KUKA KRL program: MyProgram_038().src

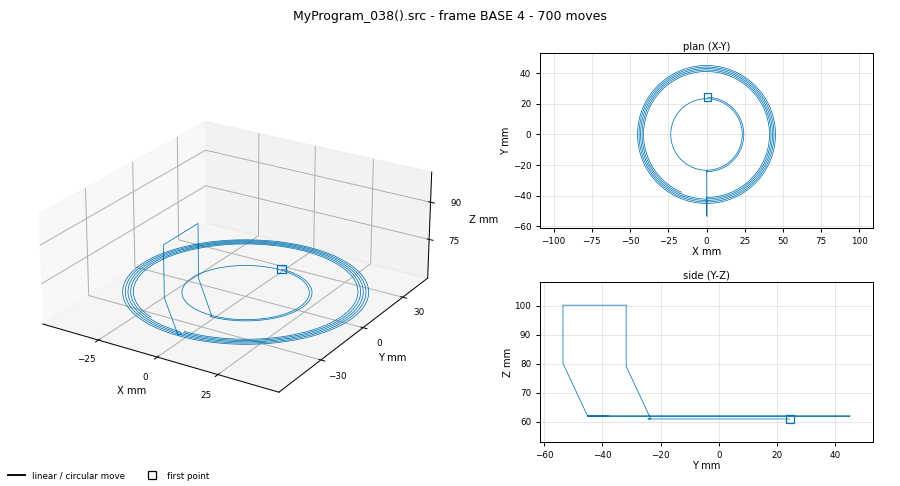
[picture p0: tool path of MyProgram_038().src in frame BASE 4, 700 of 700 moves have a stored position in this frame; points joined in program order, loops and branches not executed]
&ACCESS RVP
&REL 1
&PARAM TEMPLATE = C:\KRC\Roboter\Template\vorgabe
&PARAM EDITMASK = *
DEF MyProgram_038()
; ---- Setting reference (Base) ----
$BASE = BASE_DATA[4]

; --------------------------
; ---- Setting tool (TCP) ----
$TOOL = TOOL_DATA[3]
; --------------------------

$VEL.CP = VEL_APROX_PRINT
Startdeposition()
$VEL.CP = VEL_PRINT
LIN {X 0.6576,Y 24.378,Z 61,A 79.6841,B 24.798,C -3.2768,E1 25.0073,E2 -357.1342} C_DIS
LIN {X 2.4777,Y 24.2605,Z 61,A 75.3476,B 24.798,C -3.2762,E1 25.0194,E2 -352.7985} C_DIS
LIN {X 4.2079,Y 24.0211,Z 61,A 71.1898,B 24.7983,C -3.2745,E1 25.0308,E2 -348.6408} C_DIS
LIN {X 6.0369,Y 23.6276,Z 61,A 66.8091,B 24.7986,C -3.2723,E1 25.0427,E2 -344.261} C_DIS
LIN {X 7.8263,Y 23.0968,Z 61,A 62.2092,B 24.7992,C -3.2672,E1 25.055,E2 -339.6573} C_DIS
LIN {X 9.7348,Y 22.3594,Z 61,A 57.8843,B 24.7992,C -3.2666,E1 25.0661,E2 -335.3411} C_DIS
LIN {X 11.6331,Y 21.4331,Z 61,A 51.9674,B 24.8011,C -3.2518,E1 25.0809,E2 -329.4051} C_DIS
LIN {X 13.7357,Y 20.1506,Z 61,A 46.5226,B 24.8018,C -3.2461,E1 25.0936,E2 -323.9647} C_DIS
LIN {X 15.5109,Y 18.8183,Z 61,A 41.6965,B 24.8025,C -3.2406,E1 25.1042,E2 -319.1435} C_DIS
LIN {X 16.7453,Y 17.7285,Z 61,A 37.3106,B 24.804,C -3.2279,E1 25.1132,E2 -314.7453} C_DIS
LIN {X 18.8106,Y 15.5203,Z 61,A 30.4494,B 24.8056,C -3.2147,E1 25.1259,E2 -307.8835} C_DIS
LIN {X 20.1422,Y 13.748,Z 61,A 25.5563,B 24.8068,C -3.2054,E1 25.1338,E2 -302.992} C_DIS
LIN {X 20.9302,Y 12.5161,Z 61,A 22.3998,B 24.8075,C -3.1995,E1 25.1384,E2 -299.8377} C_DIS
LIN {X 21.6103,Y 11.3009,Z 61,A 18.8323,B 24.8089,C -3.1877,E1 25.1432,E2 -296.2609} C_DIS
LIN {X 22.463,Y 9.4933,Z 61,A 14.3404,B 24.8102,C -3.1769,E1 25.1483,E2 -291.768} C_DIS
LIN {X 23.0782,Y 7.8813,Z 61,A 10.2587,B 24.8116,C -3.165,E1 25.1522,E2 -287.6809} C_DIS
LIN {X 23.5913,Y 6.1782,Z 61,A 6.2664,B 24.8129,C -3.1548,E1 25.1552,E2 -283.6871} C_DIS
LIN {X 23.9107,Y 4.794,Z 61,A 3.2615,B 24.8136,C -3.1484,E1 25.157,E2 -280.6846} C_DIS
LIN {X 24.0965,Y 3.7504,Z 61,A 0.195,B 24.8153,C -3.1345,E1 25.1584,E2 -277.6031} C_DIS
LIN {X 24.3261,Y 1.7192,Z 61,A -4.4464,B 24.8168,C -3.1214,E1 25.1596,E2 -272.9583} C_DIS
LIN {X 24.3856,Y -0.076,Z 61,A -8.4621,B 24.8181,C -3.1105,E1 25.1597,E2 -268.9408} C_DIS
LIN {X 24.3156,Y -1.8616,Z 61,A -12.7948,B 24.8198,C -3.0959,E1 25.1591,E2 -264.5991} C_DIS
LIN {X 24.1022,Y -3.7139,Z 61,A -16.7586,B 24.8209,C -3.0869,E1 25.1576,E2 -260.6373} C_DIS
LIN {X 23.6477,Y -5.9589,Z 61,A -22.4108,B 24.8231,C -3.0672,E1 25.1543,E2 -254.9714} C_DIS
LIN {X 23.2604,Y -7.3264,Z 61,A -26.4458,B 24.8252,C -3.0494,E1 25.1509,E2 -250.9172} C_DIS
LIN {X 22.4045,Y -9.6314,Z 61,A -31.5534,B 24.8263,C -3.0395,E1 25.1457,E2 -245.8144} C_DIS
LIN {X 21.5556,Y -11.4048,Z 61,A -36.5253,B 24.8283,C -3.0224,E1 25.1394,E2 -240.8283} C_DIS
LIN {X 20.2637,Y -13.5686,Z 61,A -41.8677,B 24.8295,C -3.0122,E1 25.1315,E2 -235.4888} C_DIS
LIN {X 19.4766,Y -14.6755,Z 61,A -44.8622,B 24.8302,C -3.0059,E1 25.1265,E2 -232.4937} C_DIS
LIN {X 18.4591,Y -15.9371,Z 61,A -49.0447,B 24.8317,C -2.9922,E1 25.119,E2 -228.2982} C_DIS
LIN {X 17.1878,Y -17.3001,Z 61,A -53.3461,B 24.8328,C -2.9826,E1 25.1107,E2 -223.9923} C_DIS
LIN {X 15.9747,Y -18.4257,Z 61,A -56.7982,B 24.8333,C -2.9783,E1 25.1035,E2 -220.5439} C_DIS
LIN {X 15.0855,Y -19.1609,Z 61,A -59.5057,B 24.8339,C -2.9725,E1 25.0976,E2 -217.8329} C_DIS
LIN {X 13.9507,Y -20.0022,Z 61,A -63.1749,B 24.8351,C -2.9623,E1 25.0893,E2 -214.1524} C_DIS
LIN {X 12.5585,Y -20.9047,Z 61,A -66.515,B 24.8353,C -2.9606,E1 25.0814,E2 -210.819} C_DIS
LIN {X 11.549,Y -21.4787,Z 61,A -69.6521,B 24.8362,C -2.952,E1 25.0737,E2 -207.6705} C_DIS
LIN {X 10.141,Y -22.1785,Z 61,A -73.5285,B 24.8371,C -2.9445,E1 25.0639,E2 -203.7865} C_DIS
LIN {X 8.4683,Y -22.8694,Z 61,A -77.5795,B 24.8375,C -2.9407,E1 25.0534,E2 -199.7352} C_DIS
LIN {X 7.2197,Y -23.2934,Z 61,A -80.9229,B 24.8381,C -2.9348,E1 25.0445,E2 -196.3842} C_DIS
LIN {X 5.8698,Y -23.6699,Z 61,A -84.8468,B 24.8391,C -2.926,E1 25.0338,E2 -192.4451} C_DIS
LIN {X 3.4157,Y -24.1463,Z 61,A -89.8947,B 24.8388,C -2.9287,E1 25.0199,E2 -187.4091} C_DIS
LIN {X 1.6154,Y -24.3331,Z 61,A -94.2888,B 24.8392,C -2.9255,E1 25.0077,E2 -183.0095} C_DIS
LIN {X 0.1346,Y -24.3815,Z 61,A -96.6732,B 24.8383,C -2.9336,E1 25.0011,E2 -180.645} C_DIS
Enddeposition()
LIN {X 0.1346,Y -24.3815,Z 61,A -96.6732,B 24.8383,C -2.9336,E1 25.0011,E2 -180.645} C_DIS
Startdeposition()
$VEL.CP = VEL_PRINT
LIN {X 0.4821,Y -23.3967,Z 61,A -94.7836,B 24.8354,C -2.9592,E1 25.0065,E2 -182.5952} C_DIS
LIN {X 2.1977,Y -23.2983,Z 61,A -90.4932,B 24.8351,C -2.9619,E1 25.0185,E2 -186.8898} C_DIS
LIN {X 3.9008,Y -23.0743,Z 61,A -86.3802,B 24.8349,C -2.964,E1 25.0299,E2 -191.004} C_DIS
LIN {X 5.5815,Y -22.7263,Z 61,A -82.17,B 24.8345,C -2.9679,E1 25.0413,E2 -195.2177} C_DIS
LIN {X 7.3446,Y -22.2197,Z 61,A -77.7872,B 24.834,C -2.972,E1 25.053,E2 -199.6024} C_DIS
LIN {X 8.8729,Y -21.6544,Z 61,A -73.7272,B 24.8333,C -2.978,E1 25.0636,E2 -203.6678} C_DIS
LIN {X 10.4384,Y -20.9447,Z 61,A -69.5097,B 24.8326,C -2.9846,E1 25.0742,E2 -207.8899} C_DIS
LIN {X 11.9544,Y -20.1179,Z 61,A -65.2481,B 24.8317,C -2.9923,E1 25.0846,E2 -212.1571} C_DIS
LIN {X 13.4495,Y -19.151,Z 61,A -60.9988,B 24.8309,C -2.9996,E1 25.0944,E2 -216.4095} C_DIS
LIN {X 14.8782,Y -18.0634,Z 61,A -56.5009,B 24.8297,C -3.0099,E1 25.1043,E2 -220.9151} C_DIS
LIN {X 16.2712,Y -16.8192,Z 61,A -51.9607,B 24.8286,C -3.0201,E1 25.1136,E2 -225.4608} C_DIS
LIN {X 17.5911,Y -15.4335,Z 61,A -47.3398,B 24.8273,C -3.0309,E1 25.1223,E2 -230.087} C_DIS
LIN {X 18.7335,Y -14.0247,Z 61,A -42.9703,B 24.8261,C -3.0417,E1 25.1298,E2 -234.4614} C_DIS
LIN {X 19.7022,Y -12.6277,Z 61,A -38.7961,B 24.8248,C -3.0531,E1 25.1363,E2 -238.642} C_DIS
LIN {X 20.5911,Y -11.1195,Z 61,A -34.493,B 24.8234,C -3.0654,E1 25.1422,E2 -242.9519} C_DIS
LIN {X 21.2756,Y -9.747,Z 61,A -30.8472,B 24.8222,C -3.0752,E1 25.1465,E2 -246.6012} C_DIS
LIN {X 21.9018,Y -8.2431,Z 61,A -26.7916,B 24.8208,C -3.0878,E1 25.1507,E2 -250.6643} C_DIS
LIN {X 22.4767,Y -6.5158,Z 61,A -22.4671,B 24.8193,C -3.0999,E1 25.1543,E2 -254.9928} C_DIS
LIN {X 22.8784,Y -4.9215,Z 61,A -18.4694,B 24.8179,C -3.112,E1 25.1568,E2 -258.9961} C_DIS
LIN {X 23.1776,Y -3.2307,Z 61,A -14.2077,B 24.8163,C -3.1258,E1 25.1587,E2 -263.2653} C_DIS
LIN {X 23.3521,Y -1.5221,Z 61,A -10.0343,B 24.8148,C -3.1386,E1 25.1596,E2 -267.4442} C_DIS
LIN {X 23.3967,Y 0.4812,Z 61,A -5.2469,B 24.8131,C -3.1525,E1 25.1596,E2 -272.2363} C_DIS
LIN {X 23.2984,Y 2.1957,Z 61,A -0.9845,B 24.8115,C -3.1662,E1 25.1587,E2 -276.5057} C_DIS
LIN {X 23.0748,Y 3.8974,Z 61,A 3.1273,B 24.8101,C -3.178,E1 25.157,E2 -280.6214} C_DIS
LIN {X 22.7212,Y 5.6026,Z 61,A 7.3368,B 24.8086,C -3.1902,E1 25.1544,E2 -284.8353} C_DIS
LIN {X 22.2215,Y 7.3391,Z 61,A 11.6522,B 24.8072,C -3.2019,E1 25.1509,E2 -289.1539} C_DIS
LIN {X 21.684,Y 8.8002,Z 61,A 15.6019,B 24.8057,C -3.2142,E1 25.1469,E2 -293.1108} C_DIS
LIN {X 20.9488,Y 10.43,Z 61,A 19.8688,B 24.8044,C -3.225,E1 25.1417,E2 -297.3802} C_DIS
LIN {X 20.117,Y 11.9559,Z 61,A 24.1861,B 24.803,C -3.2367,E1 25.1358,E2 -301.703} C_DIS
LIN {X 19.0819,Y 13.547,Z 61,A 28.7529,B 24.8017,C -3.2473,E1 25.1286,E2 -306.2725} C_DIS
LIN {X 17.9987,Y 14.9561,Z 61,A 33.0946,B 24.8004,C -3.2573,E1 25.121,E2 -310.6175} C_DIS
LIN {X 16.7652,Y 16.3272,Z 61,A 37.6578,B 24.7992,C -3.2674,E1 25.1123,E2 -315.1848} C_DIS
LIN {X 15.4284,Y 17.5955,Z 61,A 42.0949,B 24.7982,C -3.2755,E1 25.1031,E2 -319.6232} C_DIS
LIN {X 14.0165,Y 18.7397,Z 61,A 46.481,B 24.7973,C -3.2827,E1 25.0935,E2 -324.0102} C_DIS
LIN {X 12.599,Y 19.7207,Z 61,A 50.7583,B 24.7964,C -3.2898,E1 25.0835,E2 -328.2902} C_DIS
LIN {X 11.0488,Y 20.6295,Z 61,A 55.0577,B 24.7958,C -3.2948,E1 25.0731,E2 -332.5889} C_DIS
LIN {X 9.4872,Y 21.3927,Z 61,A 59.3098,B 24.7952,C -3.2996,E1 25.0623,E2 -336.8416} C_DIS
LIN {X 7.8909,Y 22.0315,Z 61,A 63.4425,B 24.7948,C -3.3028,E1 25.0515,E2 -340.973} C_DIS
LIN {X 6.2392,Y 22.555,Z 61,A 67.7455,B 24.7943,C -3.3063,E1 25.04,E2 -345.2768} C_DIS
LIN {X 4.5669,Y 22.9521,Z 61,A 71.9513,B 24.7941,C -3.3083,E1 25.0285,E2 -349.4818} C_DIS
LIN {X 2.9587,Y 23.2139,Z 61,A 76.0249,B 24.7939,C -3.31,E1 25.0173,E2 -353.5558} C_DIS
LIN {X 1.1581,Y 23.3733,Z 61,A 80.3651,B 24.7939,C -3.3094,E1 25.0052,E2 -357.8926} C_DIS
LIN {X -0.4696,Y 23.397,Z 61,A 84.3727,B 24.794,C -3.3087,E1 24.994,E2 -361.8986} C_DIS
LIN {X -2.2037,Y 23.2977,Z 61,A 88.6974,B 24.7942,C -3.3074,E1 24.982,E2 -366.2221} C_DIS
LIN {X -3.9081,Y 23.073,Z 61,A 92.8279,B 24.7946,C -3.3041,E1 24.9706,E2 -370.3482} C_DIS
LIN {X -5.5911,Y 22.724,Z 61,A 97.0452,B 24.7951,C -3.3005,E1 24.9591,E2 -374.5623} C_DIS
LIN {X -7.3245,Y 22.2262,Z 61,A 101.4177,B 24.7957,C -3.2953,E1 24.9474,E2 -378.93} C_DIS
LIN {X -8.8731,Y 21.6543,Z 61,A 105.5215,B 24.7963,C -3.2905,E1 24.9368,E2 -383.0309} C_DIS
LIN {X -10.4256,Y 20.951,Z 61,A 109.7063,B 24.7971,C -3.2842,E1 24.9262,E2 -387.2115} C_DIS
LIN {X -11.9152,Y 20.1411,Z 61,A 113.9587,B 24.7979,C -3.2778,E1 24.9159,E2 -391.4609} C_DIS
LIN {X -13.4405,Y 19.1572,Z 61,A 118.3881,B 24.799,C -3.2692,E1 24.9057,E2 -395.8847} C_DIS
LIN {X -14.9859,Y 17.9739,Z 61,A 123.2373,B 24.8001,C -3.2597,E1 24.8951,E2 -400.7292} C_DIS
LIN {X -16.4031,Y 16.6906,Z 61,A 127.8701,B 24.8015,C -3.2488,E1 24.8857,E2 -405.3548} C_DIS
LIN {X -17.6037,Y 15.419,Z 61,A 132.2093,B 24.8027,C -3.2387,E1 24.8776,E2 -409.6891} C_DIS
LIN {X -18.7457,Y 14.0085,Z 61,A 136.6265,B 24.8041,C -3.2271,E1 24.87,E2 -414.0995} C_DIS
LIN {X -19.7705,Y 12.5213,Z 61,A 141.1344,B 24.8055,C -3.2156,E1 24.8631,E2 -418.6023} C_DIS
LIN {X -20.6499,Y 11.0105,Z 61,A 145.3779,B 24.807,C -3.2033,E1 24.8573,E2 -422.8388} C_DIS
LIN {X -21.3982,Y 9.4747,Z 61,A 149.5929,B 24.8085,C -3.1913,E1 24.8524,E2 -427.048} C_DIS
LIN {X -22.0333,Y 7.886,Z 61,A 153.7349,B 24.81,C -3.1786,E1 24.8483,E2 -431.1828} C_DIS
LIN {X -22.5504,Y 6.2556,Z 61,A 158.034,B 24.8115,C -3.1664,E1 24.8449,E2 -435.4775} C_DIS
LIN {X -22.9461,Y 4.5961,Z 61,A 162.3444,B 24.8129,C -3.1541,E1 24.8423,E2 -439.7839} C_DIS
LIN {X -23.2409,Y 2.7382,Z 61,A 166.9452,B 24.8146,C -3.1398,E1 24.8405,E2 -444.3777} C_DIS
LIN {X -23.3851,Y 0.8879,Z 61,A 171.5741,B 24.8163,C -3.126,E1 24.8398,E2 -449.0015} C_DIS
LIN {X -23.3863,Y -0.8572,Z 61,A 175.7875,B 24.8179,C -3.1124,E1 24.84,E2 -453.2077} C_DIS
LIN {X -23.2682,Y -2.4958,Z 61,A 179.9115,B 24.8193,C -3.1005,E1 24.8411,E2 -457.3279} C_DIS
LIN {X -23.0063,Y -4.2856,Z 61,A -175.7162,B 24.8209,C -3.0868,E1 24.8431,E2 -461.6933} C_DIS
LIN {X -22.6518,Y -5.8766,Z 61,A -171.6959,B 24.8222,C -3.0751,E1 24.8457,E2 -465.709} C_DIS
LIN {X -22.1592,Y -7.5238,Z 61,A -167.406,B 24.8236,C -3.0632,E1 24.8494,E2 -469.9952} C_DIS
LIN {X -21.5076,Y -9.2238,Z 61,A -162.8218,B 24.825,C -3.0514,E1 24.8542,E2 -474.5765} C_DIS
LIN {X -20.9375,Y -10.4529,Z 61,A -159.6322,B 24.8261,C -3.0418,E1 24.8581,E2 -477.7603} C_DIS
LIN {X -20.1157,Y -11.9582,Z 61,A -155.3205,B 24.8273,C -3.0314,E1 24.8641,E2 -482.0699} C_DIS
LIN {X -19.0827,Y -13.5458,Z 61,A -150.6719,B 24.8286,C -3.0201,E1 24.8713,E2 -486.7145} C_DIS
LIN {X -18.0046,Y -14.9489,Z 61,A -146.3168,B 24.8297,C -3.0103,E1 24.8789,E2 -491.0664} C_DIS
LIN {X -16.7508,Y -16.3422,Z 61,A -141.7569,B 24.8308,C -3.0004,E1 24.8876,E2 -495.6225} C_DIS
LIN {X -15.4267,Y -17.597,Z 61,A -137.2275,B 24.8317,C -2.9921,E1 24.897,E2 -500.1504} C_DIS
LIN {X -14.0182,Y -18.7384,Z 61,A -132.8261,B 24.8326,C -2.9841,E1 24.9067,E2 -504.5489} C_DIS
LIN {X -12.5345,Y -19.762,Z 61,A -128.3797,B 24.8334,C -2.9776,E1 24.917,E2 -508.9943} C_DIS
LIN {X -11.0359,Y -20.6365,Z 61,A -124.1142,B 24.834,C -2.9721,E1 24.9274,E2 -513.259} C_DIS
LIN {X -9.4793,Y -21.3962,Z 61,A -119.8794,B 24.8345,C -2.9673,E1 24.9381,E2 -517.493} C_DIS
LIN {X -7.8834,Y -22.0343,Z 61,A -115.7407,B 24.835,C -2.9631,E1 24.9489,E2 -521.6302} C_DIS
LIN {X -6.2449,Y -22.5534,Z 61,A -111.4444,B 24.8352,C -2.9609,E1 24.9604,E2 -525.9284} C_DIS
LIN {X -4.5731,Y -22.9509,Z 61,A -107.2323,B 24.8355,C -2.959,E1 24.9719,E2 -530.1414} C_DIS
LIN {X -2.9659,Y -23.213,Z 61,A -103.1543,B 24.8355,C -2.9589,E1 24.9832,E2 -534.2224} C_DIS
LIN {X -1.147,Y -23.3739,Z 61,A -98.7713,B 24.8355,C -2.9582,E1 24.9954,E2 -538.6054} C_DIS
LIN {X 0.1301,Y -23.3984,Z 61,A -96.7291,B 24.8364,C -2.9502,E1 25.0011,E2 -540.6285} C_DIS
Enddeposition()
LIN {X 0.1399,Y -25.5114,Z 65.5315,A -96.7152,B 24.8371,C -2.9443,E1 25.0011,E2 -540.6285} C_DIS
LIN {X 0.1693,Y -31.8506,Z 79.1262,A -96.6781,B 24.8388,C -2.9287,E1 25.0011,E2 -540.6285} C_DIS
LIN {X 0.1693,Y -31.8506,Z 100.1262,A -97.0269,B 24.8222,C -3.0752,E1 25.0011,E2 -540.6285} C_DIS
LIN {X 0.2145,Y -53.5807,Z 100.1262,A -96.4159,B 24.8624,C -2.7068,E1 25.0003,E2 -540.3627} C_DIS
LIN {X 0.2145,Y -53.5807,Z 80.1262,A -96.0843,B 24.8763,C -2.5674,E1 25.0003,E2 -540.3627} C_DIS
LIN {X 0.2145,Y -47.2414,Z 66.5315,A -96.118,B 24.8749,C -2.5815,E1 25.0003,E2 -540.3627} C_DIS
LIN {X 0.2145,Y -45.1283,Z 62,A -96.1307,B 24.8744,C -2.5869,E1 25.0003,E2 -540.3627} C_DIS
Startdeposition()
$VEL.CP = VEL_PRINT
LIN {X 1.6717,Y -45.1007,Z 62,A -93.3413,B 24.8729,C -2.6023,E1 25.0082,E2 -543.1881} C_DIS
LIN {X 3.8826,Y -44.9643,Z 62,A -90.5016,B 24.8727,C -2.604,E1 25.0161,E2 -546.0305} C_DIS
LIN {X 6.0842,Y -44.7196,Z 62,A -87.7329,B 24.8726,C -2.605,E1 25.0238,E2 -548.7995} C_DIS
LIN {X 8.2712,Y -44.3672,Z 62,A -84.9157,B 24.8724,C -2.6073,E1 25.0315,E2 -551.619} C_DIS
LIN {X 10.428,Y -43.9104,Z 62,A -82.1224,B 24.8721,C -2.6097,E1 25.0392,E2 -554.4144} C_DIS
LIN {X 12.5801,Y -43.3429,Z 62,A -79.3131,B 24.8719,C -2.6124,E1 25.0467,E2 -557.2255} C_DIS
LIN {X 14.6818,Y -42.6769,Z 62,A -76.512,B 24.8715,C -2.6158,E1 25.0542,E2 -560.0294} C_DIS
LIN {X 16.7582,Y -41.905,Z 62,A -73.7082,B 24.8712,C -2.6195,E1 25.0615,E2 -562.8357} C_DIS
LIN {X 18.8037,Y -41.0278,Z 62,A -70.892,B 24.8708,C -2.6235,E1 25.0687,E2 -565.6545} C_DIS
LIN {X 20.7849,Y -40.0607,Z 62,A -68.0934,B 24.8703,C -2.628,E1 25.0756,E2 -568.4562} C_DIS
LIN {X 22.7346,Y -38.9872,Z 62,A -65.2886,B 24.8699,C -2.6326,E1 25.0825,E2 -571.2636} C_DIS
LIN {X 24.6202,Y -37.8247,Z 62,A -62.488,B 24.8694,C -2.6377,E1 25.0891,E2 -574.0671} C_DIS
LIN {X 26.438,Y -36.5773,Z 62,A -59.6921,B 24.8688,C -2.6432,E1 25.0955,E2 -576.8664} C_DIS
LIN {X 28.201,Y -35.236,Z 62,A -56.8931,B 24.8682,C -2.6489,E1 25.1016,E2 -579.6686} C_DIS
LIN {X 29.8959,Y -33.8098,Z 62,A -54.1044,B 24.8677,C -2.6547,E1 25.1075,E2 -582.4602} C_DIS
LIN {X 31.5264,Y -32.2948,Z 62,A -51.2936,B 24.867,C -2.661,E1 25.1132,E2 -585.2743} C_DIS
LIN {X 33.073,Y -30.7089,Z 62,A -48.5064,B 24.8664,C -2.6674,E1 25.1186,E2 -588.0646} C_DIS
LIN {X 34.5333,Y -29.0572,Z 62,A -45.7138,B 24.8657,C -2.6744,E1 25.1237,E2 -590.8609} C_DIS
LIN {X 35.9175,Y -27.3277,Z 62,A -42.918,B 24.865,C -2.6814,E1 25.1285,E2 -593.6602} C_DIS
LIN {X 37.221,Y -25.5237,Z 62,A -40.1096,B 24.8642,C -2.6887,E1 25.133,E2 -596.4722} C_DIS
LIN {X 38.4231,Y -23.6756,Z 62,A -37.328,B 24.8635,C -2.6962,E1 25.1372,E2 -599.2574} C_DIS
LIN {X 39.5435,Y -21.7525,Z 62,A -34.5206,B 24.8627,C -2.7038,E1 25.141,E2 -602.0684} C_DIS
LIN {X 40.5632,Y -19.786,Z 62,A -31.7266,B 24.8619,C -2.7117,E1 25.1445,E2 -604.8661} C_DIS
LIN {X 41.4852,Y -17.7718,Z 62,A -28.9427,B 24.8611,C -2.7195,E1 25.1477,E2 -607.6532} C_DIS
LIN {X 42.3037,Y -15.7247,Z 62,A -26.1532,B 24.8603,C -2.7277,E1 25.1505,E2 -610.4468} C_DIS
LIN {X 43.0274,Y -13.62,Z 62,A -23.3563,B 24.8594,C -2.7358,E1 25.1529,E2 -613.2469} C_DIS
LIN {X 43.6413,Y -11.5025,Z 62,A -20.5675,B 24.8586,C -2.7442,E1 25.155,E2 -616.0397} C_DIS
LIN {X 44.1552,Y -9.337,Z 62,A -17.7713,B 24.8577,C -2.7525,E1 25.1567,E2 -618.8391} C_DIS
LIN {X 44.5586,Y -7.1695,Z 62,A -14.973,B 24.8568,C -2.7612,E1 25.1581,E2 -621.6417} C_DIS
LIN {X 44.8578,Y -4.9641,Z 62,A -12.1768,B 24.8559,C -2.7696,E1 25.159,E2 -624.4411} C_DIS
LIN {X 45.0473,Y -2.757,Z 62,A -9.3942,B 24.8551,C -2.7778,E1 25.1596,E2 -627.2268} C_DIS
LIN {X 45.1183,Y -1.0971,Z 62,A -7.1841,B 24.8542,C -2.7864,E1 25.1598,E2 -629.4439} C_DIS
LIN {X 45.1178,Y 1.1181,Z 62,A -4.498,B 24.8535,C -2.7928,E1 25.1597,E2 -632.1293} C_DIS
LIN {X 45.0094,Y 3.3201,Z 62,A -1.7185,B 24.8526,C -2.8012,E1 25.1592,E2 -634.9121} C_DIS
LIN {X 44.7923,Y 5.5246,Z 62,A 1.0837,B 24.8517,C -2.8097,E1 25.1583,E2 -637.7179} C_DIS
LIN {X 44.4654,Y 7.7261,Z 62,A 3.9908,B 24.8506,C -2.8199,E1 25.157,E2 -640.632} C_DIS
LIN {X 44.0327,Y 9.8986,Z 62,A 6.6733,B 24.85,C -2.826,E1 25.1555,E2 -643.3132} C_DIS
LIN {X 43.494,Y 12.0473,Z 62,A 9.457,B 24.8491,C -2.8338,E1 25.1535,E2 -646.0995} C_DIS
LIN {X 42.8075,Y 14.2943,Z 62,A 12.3147,B 24.8484,C -2.8403,E1 25.151,E2 -648.9562} C_DIS
LIN {X 42.1037,Y 16.2524,Z 62,A 15.0449,B 24.8475,C -2.8494,E1 25.1484,E2 -651.693} C_DIS
LIN {X 41.2555,Y 18.2988,Z 62,A 17.8491,B 24.8466,C -2.8572,E1 25.1453,E2 -654.5} C_DIS
LIN {X 40.3127,Y 20.2917,Z 62,A 20.6475,B 24.8458,C -2.8648,E1 25.1419,E2 -657.3015} C_DIS
LIN {X 39.2633,Y 22.2544,Z 62,A 23.43,B 24.8451,C -2.8715,E1 25.1381,E2 -660.0853} C_DIS
LIN {X 38.1297,Y 24.1453,Z 62,A 26.2223,B 24.8443,C -2.8786,E1 25.134,E2 -662.8801} C_DIS
LIN {X 36.8929,Y 25.9957,Z 62,A 29.0322,B 24.8436,C -2.8853,E1 25.1296,E2 -665.6922} C_DIS
LIN {X 35.5729,Y 27.7747,Z 62,A 31.8295,B 24.8429,C -2.8917,E1 25.1248,E2 -668.4912} C_DIS
LIN {X 34.1741,Y 29.4788,Z 62,A 34.6141,B 24.8422,C -2.8978,E1 25.1198,E2 -671.2776} C_DIS
LIN {X 32.6792,Y 31.1277,Z 62,A 37.4165,B 24.8416,C -2.9034,E1 25.1145,E2 -674.0812} C_DIS
LIN {X 31.1125,Y 32.6937,Z 62,A 40.2159,B 24.841,C -2.909,E1 25.1089,E2 -676.882} C_DIS
LIN {X 29.4788,Y 34.1741,Z 62,A 43.0122,B 24.8404,C -2.9143,E1 25.103,E2 -679.6799} C_DIS
LIN {X 27.7581,Y 35.5858,Z 62,A 45.8169,B 24.8399,C -2.9191,E1 25.0969,E2 -682.4853} C_DIS
LIN {X 25.9872,Y 36.899,Z 62,A 48.6244,B 24.8394,C -2.9239,E1 25.0906,E2 -685.2944} C_DIS
LIN {X 24.1364,Y 38.1352,Z 62,A 51.4212,B 24.8389,C -2.9278,E1 25.084,E2 -688.0912} C_DIS
LIN {X 22.2453,Y 39.2685,Z 62,A 54.2303,B 24.8385,C -2.9319,E1 25.0772,E2 -690.9015} C_DIS
LIN {X 20.2917,Y 40.3127,Z 62,A 57.0342,B 24.8381,C -2.9353,E1 25.0703,E2 -693.7058} C_DIS
LIN {X 18.2796,Y 41.264,Z 62,A 59.8435,B 24.8378,C -2.9382,E1 25.0631,E2 -696.5149} C_DIS
LIN {X 16.2329,Y 42.1113,Z 62,A 62.7796,B 24.8372,C -2.943,E1 25.0555,E2 -699.4558} C_DIS
LIN {X 14.147,Y 42.857,Z 62,A 65.4473,B 24.8372,C -2.943,E1 25.0485,E2 -702.1182} C_DIS
LIN {X 11.9926,Y 43.5089,Z 62,A 68.2784,B 24.8371,C -2.9445,E1 25.0409,E2 -704.9481} C_DIS
LIN {X 9.8884,Y 44.0351,Z 62,A 71.0705,B 24.8368,C -2.9466,E1 25.0333,E2 -707.7412} C_DIS
LIN {X 7.7054,Y 44.469,Z 62,A 73.8747,B 24.8368,C -2.9473,E1 25.0256,E2 -710.544} C_DIS
LIN {X 5.5246,Y 44.7923,Z 62,A 76.6915,B 24.8367,C -2.9482,E1 25.0178,E2 -713.3606} C_DIS
LIN {X 3.3201,Y 45.0094,Z 62,A 79.4938,B 24.8367,C -2.9482,E1 25.01,E2 -716.1615} C_DIS
LIN {X 1.0971,Y 45.1183,Z 62,A 82.3203,B 24.8367,C -2.9481,E1 25.0021,E2 -718.9867} C_DIS
LIN {X -1.1181,Y 45.1178,Z 62,A 85.1244,B 24.8367,C -2.9473,E1 24.9943,E2 -721.7891} C_DIS
LIN {X -3.3201,Y 45.0094,Z 62,A 87.9358,B 24.8369,C -2.9464,E1 24.9865,E2 -724.5994} C_DIS
LIN {X -5.5246,Y 44.7923,Z 62,A 90.7615,B 24.837,C -2.9451,E1 24.9786,E2 -727.4236} C_DIS
LIN {X -7.7261,Y 44.4654,Z 62,A 93.5725,B 24.8372,C -2.9429,E1 24.9709,E2 -730.2321} C_DIS
LIN {X -9.8986,Y 44.0327,Z 62,A 96.4002,B 24.8375,C -2.9408,E1 24.9632,E2 -733.0581} C_DIS
LIN {X -12.0473,Y 43.494,Z 62,A 99.2091,B 24.8378,C -2.938,E1 24.9556,E2 -735.8645} C_DIS
LIN {X -14.1669,Y 42.8505,Z 62,A 102.0387,B 24.8381,C -2.935,E1 24.9481,E2 -738.6922} C_DIS
LIN {X -16.2524,Y 42.1037,Z 62,A 104.8498,B 24.8385,C -2.9314,E1 24.9407,E2 -741.5004} C_DIS
LIN {X -18.2892,Y 41.2598,Z 62,A 107.6677,B 24.8389,C -2.9278,E1 24.9335,E2 -744.3161} C_DIS
LIN {X -20.2917,Y 40.3127,Z 62,A 110.4904,B 24.8394,C -2.9235,E1 24.9264,E2 -747.136} C_DIS
LIN {X -22.2544,Y 39.2633,Z 62,A 113.3272,B 24.8399,C -2.9189,E1 24.9195,E2 -749.97} C_DIS
LIN {X -24.1453,Y 38.1297,Z 62,A 116.138,B 24.8404,C -2.914,E1 24.9128,E2 -752.7779} C_DIS
LIN {X -25.9957,Y 36.8929,Z 62,A 118.9765,B 24.841,C -2.9087,E1 24.9063,E2 -755.6133} C_DIS
LIN {X -27.8059,Y 35.5482,Z 62,A 121.8172,B 24.8417,C -2.9026,E1 24.9,E2 -758.4496} C_DIS
LIN {X -29.4867,Y 34.1672,Z 62,A 124.6287,B 24.8423,C -2.8972,E1 24.894,E2 -761.2592} C_DIS
LIN {X -31.1201,Y 32.6865,Z 62,A 127.4426,B 24.843,C -2.8911,E1 24.8882,E2 -764.0698} C_DIS
LIN {X -32.6865,Y 31.1201,Z 62,A 130.2705,B 24.8437,C -2.8846,E1 24.8827,E2 -766.8943} C_DIS
LIN {X -34.1741,Y 29.4788,Z 62,A 133.2317,B 24.8442,C -2.8795,E1 24.8773,E2 -769.8567} C_DIS
LIN {X -35.799,Y 27.4814,Z 62,A 136.4743,B 24.8452,C -2.8708,E1 24.8717,E2 -773.0937} C_DIS
LIN {X -37.221,Y 25.5237,Z 62,A 139.4692,B 24.8462,C -2.8616,E1 24.8669,E2 -776.0813} C_DIS
LIN {X -38.4285,Y 23.6666,Z 62,A 142.2997,B 24.847,C -2.8541,E1 24.8626,E2 -778.9082} C_DIS
LIN {X -39.5385,Y 21.7618,Z 62,A 145.1268,B 24.8478,C -2.8465,E1 24.8588,E2 -781.732} C_DIS
LIN {X -40.5587,Y 19.7955,Z 62,A 147.9579,B 24.8486,C -2.8386,E1 24.8552,E2 -784.5595} C_DIS
LIN {X -41.4853,Y 17.7719,Z 62,A 150.7979,B 24.8495,C -2.8305,E1 24.852,E2 -787.3956} C_DIS
LIN {X -42.3037,Y 15.7247,Z 62,A 153.6216,B 24.8504,C -2.8224,E1 24.8492,E2 -790.2158} C_DIS
LIN {X -43.0274,Y 13.62,Z 62,A 156.4576,B 24.8513,C -2.8139,E1 24.8467,E2 -793.0478} C_DIS
LIN {X -43.6439,Y 11.4923,Z 62,A 159.29,B 24.8521,C -2.8056,E1 24.8446,E2 -795.8766} C_DIS
LIN {X -44.1552,Y 9.337,Z 62,A 162.1226,B 24.853,C -2.7971,E1 24.8429,E2 -798.7055} C_DIS
LIN {X -44.5586,Y 7.1695,Z 62,A 164.9613,B 24.8539,C -2.7888,E1 24.8415,E2 -801.5414} C_DIS
LIN {X -44.8578,Y 4.9641,Z 62,A 167.7981,B 24.8548,C -2.7801,E1 24.8405,E2 -804.3742} C_DIS
LIN {X -45.0468,Y 2.7675,Z 62,A 170.6175,B 24.8557,C -2.7716,E1 24.84,E2 -807.1902} C_DIS
LIN {X -45.1295,Y 0.3893,Z 62,A 173.5317,B 24.8568,C -2.7608,E1 24.8398,E2 -810.0961} C_DIS
LIN {X -45.1007,Y -1.6717,Z 62,A 176.2968,B 24.8575,C -2.7544,E1 24.84,E2 -812.8627} C_DIS
LIN {X -44.9643,Y -3.8826,Z 62,A 179.1295,B 24.8584,C -2.7459,E1 24.8406,E2 -815.692} C_DIS
LIN {X -44.7196,Y -6.0842,Z 62,A -178.0478,B 24.8593,C -2.7374,E1 24.8415,E2 -818.5112} C_DIS
LIN {X -44.3672,Y -8.2712,Z 62,A -175.2057,B 24.8601,C -2.7292,E1 24.8429,E2 -821.3506} C_DIS
LIN {X -43.9104,Y -10.428,Z 62,A -172.3871,B 24.8609,C -2.721,E1 24.8446,E2 -824.1661} C_DIS
LIN {X -43.3429,Y -12.5801,Z 62,A -169.5517,B 24.8618,C -2.7128,E1 24.8467,E2 -826.9982} C_DIS
LIN {X -42.6769,Y -14.6818,Z 62,A -166.724,B 24.8626,C -2.705,E1 24.8492,E2 -829.8235} C_DIS
LIN {X -41.905,Y -16.7582,Z 62,A -163.8931,B 24.8634,C -2.6972,E1 24.852,E2 -832.6518} C_DIS
LIN {X -41.0278,Y -18.8037,Z 62,A -161.0492,B 24.8642,C -2.6896,E1 24.8553,E2 -835.4931} C_DIS
LIN {X -40.0607,Y -20.7849,Z 62,A -158.2227,B 24.8649,C -2.6824,E1 24.8588,E2 -838.3175} C_DIS
LIN {X -38.9872,Y -22.7346,Z 62,A -155.3896,B 24.8656,C -2.6751,E1 24.8627,E2 -841.1479} C_DIS
LIN {X -37.8247,Y -24.6202,Z 62,A -152.5606,B 24.8663,C -2.6682,E1 24.8669,E2 -843.9748} C_DIS
LIN {X -36.5773,Y -26.438,Z 62,A -149.6444,B 24.8668,C -2.6629,E1 24.8716,E2 -846.8927} C_DIS
LIN {X -35.0844,Y -28.388,Z 62,A -146.8015,B 24.8679,C -2.652,E1 24.8765,E2 -849.723} C_DIS
LIN {X -33.8098,Y -29.8959,Z 62,A -144.0911,B 24.8682,C -2.6491,E1 24.8815,E2 -852.4388} C_DIS
LIN {X -32.2948,Y -31.5264,Z 62,A -141.2516,B 24.8688,C -2.6433,E1 24.8869,E2 -855.2768} C_DIS
LIN {X -30.7089,Y -33.073,Z 62,A -138.4359,B 24.8694,C -2.6378,E1 24.8926,E2 -858.0908} C_DIS
LIN {X -29.0572,Y -34.5333,Z 62,A -135.615,B 24.8698,C -2.6328,E1 24.8986,E2 -860.9108} C_DIS
LIN {X -27.3277,Y -35.9175,Z 62,A -132.7911,B 24.8703,C -2.628,E1 24.9048,E2 -863.7337} C_DIS
LIN {X -25.5237,Y -37.221,Z 62,A -129.9548,B 24.8708,C -2.6236,E1 24.9113,E2 -866.5692} C_DIS
LIN {X -23.6756,Y -38.4231,Z 62,A -127.1459,B 24.8712,C -2.6196,E1 24.9179,E2 -869.3775} C_DIS
LIN {X -21.7525,Y -39.5435,Z 62,A -124.3115,B 24.8715,C -2.6159,E1 24.9248,E2 -872.2114} C_DIS
LIN {X -19.7817,Y -40.5653,Z 62,A -121.4893,B 24.8718,C -2.6126,E1 24.9318,E2 -875.0332} C_DIS
LIN {X -17.7718,Y -41.4852,Z 62,A -118.6814,B 24.8721,C -2.6096,E1 24.939,E2 -877.8407} C_DIS
LIN {X -15.7247,Y -42.3037,Z 62,A -115.8667,B 24.8724,C -2.6073,E1 24.9464,E2 -880.6558} C_DIS
LIN {X -13.62,Y -43.0274,Z 62,A -113.0453,B 24.8726,C -2.605,E1 24.9538,E2 -883.4771} C_DIS
LIN {X -11.5025,Y -43.6413,Z 62,A -110.2328,B 24.8727,C -2.6035,E1 24.9614,E2 -886.2904} C_DIS
LIN {X -9.337,Y -44.1552,Z 62,A -107.4137,B 24.8729,C -2.6021,E1 24.9691,E2 -889.1097} C_DIS
LIN {X -7.0449,Y -44.5778,Z 62,A -104.5432,B 24.8731,C -2.5998,E1 24.977,E2 -891.9777} C_DIS
LIN {X -4.9641,Y -44.8578,Z 62,A -101.7759,B 24.873,C -2.601,E1 24.9847,E2 -894.7496} C_DIS
LIN {X -2.757,Y -45.0473,Z 62,A -98.9732,B 24.873,C -2.6008,E1 24.9925,E2 -897.553} C_DIS
LIN {X -0.5538,Y -45.1283,Z 62,A -96.1652,B 24.873,C -2.6014,E1 25.0003,E2 -900.3627} C_DIS
LIN {X -0.5538,Y -45.1283,Z 62,A -96.1652,B 24.873,C -2.6014,E1 25.0003,E2 -900.3627} C_DIS
Enddeposition()
LIN {X 0.2247,Y -44.1474,Z 62,A -96.7459,B 24.8736,C -2.5944,E1 24.9986,E2 -899.7654} C_DIS
Startdeposition()
$VEL.CP = VEL_PRINT
LIN {X -2.4295,Y -44.0843,Z 62,A -99.5697,B 24.8728,C -2.6033,E1 24.9908,E2 -896.9623} C_DIS
LIN {X -4.1306,Y -43.9576,Z 62,A -102.3148,B 24.8735,C -2.5955,E1 24.9831,E2 -894.1972} C_DIS
LIN {X -6.6902,Y -43.6414,Z 62,A -105.5217,B 24.8733,C -2.5982,E1 24.9743,E2 -890.9943} C_DIS
LIN {X -8.8949,Y -43.2459,Z 62,A -108.6267,B 24.8734,C -2.5964,E1 24.9657,E2 -887.8816} C_DIS
LIN {X -11.2172,Y -42.7031,Z 62,A -111.2278,B 24.8726,C -2.6051,E1 24.9587,E2 -885.2976} C_DIS
LIN {X -12.8054,Y -42.2542,Z 62,A -113.854,B 24.8731,C -2.5996,E1 24.9516,E2 -882.6541} C_DIS
LIN {X -15.1666,Y -41.4645,Z 62,A -117.0629,B 24.8728,C -2.6026,E1 24.9432,E2 -879.446} C_DIS
LIN {X -17.7622,Y -40.4209,Z 62,A -120.1335,B 24.8717,C -2.614,E1 24.9353,E2 -876.3956} C_DIS
LIN {X -19.6434,Y -39.5407,Z 62,A -123.6319,B 24.8725,C -2.6061,E1 24.9264,E2 -872.8694} C_DIS
LIN {X -21.8948,Y -38.3401,Z 62,A -126.5281,B 24.8715,C -2.616,E1 24.9194,E2 -869.9886} C_DIS
LIN {X -23.5815,Y -37.3268,Z 62,A -129.1631,B 24.8712,C -2.6186,E1 24.9131,E2 -867.3516} C_DIS
LIN {X -25.1222,Y -36.3071,Z 62,A -131.6956,B 24.8711,C -2.6206,E1 24.9073,E2 -864.8154} C_DIS
LIN {X -27.1026,Y -34.8542,Z 62,A -134.8849,B 24.8705,C -2.6261,E1 24.9002,E2 -861.6276} C_DIS
LIN {X -29.0006,Y -33.2911,Z 62,A -138.1447,B 24.87,C -2.6311,E1 24.8932,E2 -858.3672} C_DIS
LIN {X -30.5249,Y -31.8996,Z 62,A -140.8545,B 24.8695,C -2.636,E1 24.8877,E2 -855.658} C_DIS
LIN {X -32.3758,Y -30.0198,Z 62,A -144.2991,B 24.8688,C -2.643,E1 24.8811,E2 -852.2152} C_DIS
LIN {X -34.108,Y -28.0362,Z 62,A -147.6279,B 24.868,C -2.6518,E1 24.8751,E2 -848.8921} C_DIS
LIN {X -35.6435,Y -26.0551,Z 62,A -150.9329,B 24.8673,C -2.6588,E1 24.8695,E2 -845.5882} C_DIS
LIN {X -37.0239,Y -24.0545,Z 62,A -154.0824,B 24.8665,C -2.6667,E1 24.8646,E2 -842.4418} C_DIS
LIN {X -38.2479,Y -22.0552,Z 62,A -157.1606,B 24.8657,C -2.6741,E1 24.8602,E2 -839.3655} C_DIS
LIN {X -39.3052,Y -20.1104,Z 62,A -160.2764,B 24.8652,C -2.6789,E1 24.8562,E2 -836.2445} C_DIS
LIN {X -40.4887,Y -17.6066,Z 62,A -163.7713,B 24.8641,C -2.69,E1 24.8522,E2 -832.757} C_DIS
LIN {X -41.3651,Y -15.4371,Z 62,A -166.7149,B 24.8631,C -2.6998,E1 24.8492,E2 -829.8202} C_DIS
LIN {X -42.2014,Y -12.9741,Z 62,A -170.0451,B 24.8621,C -2.7101,E1 24.8463,E2 -826.4958} C_DIS
LIN {X -42.8594,Y -10.6027,Z 62,A -173.189,B 24.861,C -2.7202,E1 24.8441,E2 -823.3576} C_DIS
LIN {X -43.3646,Y -8.297,Z 62,A -176.3189,B 24.8602,C -2.7287,E1 24.8423,E2 -820.2296} C_DIS
LIN {X -43.719,Y -6.1625,Z 62,A -179.1102,B 24.8593,C -2.7375,E1 24.8411,E2 -817.4427} C_DIS
LIN {X -44.0134,Y -3.4853,Z 62,A 176.9209,B 24.8587,C -2.7428,E1 24.8401,E2 -813.4627} C_DIS
LIN {X -44.1374,Y -1.1268,Z 62,A 174.2044,B 24.8573,C -2.7564,E1 24.8398,E2 -810.7624} C_DIS
LIN {X -44.1357,Y 1.1802,Z 62,A 171.2539,B 24.8563,C -2.7663,E1 24.8398,E2 -807.8178} C_DIS
LIN {X -44.0263,Y 3.3243,Z 62,A 168.4616,B 24.8554,C -2.775,E1 24.8404,E2 -805.0294} C_DIS
LIN {X -43.8005,Y 5.5547,Z 62,A 165.5693,B 24.8544,C -2.7843,E1 24.8413,E2 -802.1422} C_DIS
LIN {X -43.4395,Y 7.896,Z 62,A 162.2642,B 24.8537,C -2.7912,E1 24.8428,E2 -798.8339} C_DIS
LIN {X -42.6766,Y 11.3172,Z 62,A 157.078,B 24.8529,C -2.798,E1 24.8462,E2 -793.6336} C_DIS
LIN {X -41.9192,Y 13.8611,Z 62,A 154.3866,B 24.8509,C -2.8172,E1 24.8485,E2 -790.9726} C_DIS
LIN {X -41.1229,Y 16.0699,Z 62,A 151.0997,B 24.8502,C -2.8235,E1 24.8517,E2 -787.6824} C_DIS
LIN {X -40.2479,Y 18.1502,Z 62,A 148.4392,B 24.849,C -2.8353,E1 24.8546,E2 -785.0354} C_DIS
LIN {X -39.4291,Y 19.868,Z 62,A 145.7174,B 24.8485,C -2.8395,E1 24.858,E2 -782.3089} C_DIS
LIN {X -38.2925,Y 21.9775,Z 62,A 142.6263,B 24.8476,C -2.8485,E1 24.8622,E2 -779.2232} C_DIS
LIN {X -37.0899,Y 23.9516,Z 62,A 139.1662,B 24.8473,C -2.8513,E1 24.8674,E2 -775.7522} C_DIS
LIN {X -34.8259,Y 27.1393,Z 62,A 134.7628,B 24.8449,C -2.8728,E1 24.8746,E2 -771.3788} C_DIS
LIN {X -32.9685,Y 29.367,Z 62,A 130.1834,B 24.8449,C -2.8723,E1 24.883,E2 -766.7776} C_DIS
LIN {X -30.6331,Y 31.7953,Z 62,A 125.935,B 24.8437,C -2.8841,E1 24.8913,E2 -762.5394} C_DIS
LIN {X -27.7378,Y 34.3504,Z 62,A 121.4148,B 24.8418,C -2.9012,E1 24.9009,E2 -758.0424} C_DIS
LIN {X -25.9309,Y 35.7344,Z 62,A 118.227,B 24.8415,C -2.9042,E1 24.908,E2 -754.8504} C_DIS
LIN {X -24.0027,Y 37.0572,Z 62,A 114.9889,B 24.8412,C -2.9074,E1 24.9156,E2 -751.6093} C_DIS
LIN {X -20.9899,Y 38.8427,Z 62,A 110.9445,B 24.8396,C -2.9217,E1 24.9253,E2 -747.587} C_DIS
LIN {X -19.0828,Y 39.8143,Z 62,A 107.8124,B 24.8396,C -2.9214,E1 24.9332,E2 -744.4459} C_DIS
LIN {X -16.9934,Y 40.7502,Z 62,A 104.0493,B 24.8403,C -2.9152,E1 24.9429,E2 -740.6594} C_DIS
LIN {X -14.3563,Y 41.7528,Z 62,A 100.8102,B 24.8392,C -2.9252,E1 24.9514,E2 -737.4378} C_DIS
LIN {X -11.2523,Y 42.6922,Z 62,A 97.1317,B 24.8379,C -2.9368,E1 24.9612,E2 -733.7811} C_DIS
LIN {X -8.8221,Y 43.2608,Z 62,A 94.2728,B 24.837,C -2.9449,E1 24.969,E2 -730.9377} C_DIS
LIN {X -7.1087,Y 43.5755,Z 62,A 91.5538,B 24.8376,C -2.9401,E1 24.9765,E2 -728.2047} C_DIS
LIN {X -4.5241,Y 43.9188,Z 62,A 88.084,B 24.8375,C -2.9408,E1 24.9861,E2 -724.7343} C_DIS
LIN {X -1.9287,Y 44.109,Z 62,A 84.5117,B 24.8376,C -2.9393,E1 24.9961,E2 -721.1573} C_DIS
LIN {X 0.8225,Y 44.1435,Z 62,A 81.189,B 24.8372,C -2.9435,E1 25.0053,E2 -717.8449} C_DIS
LIN {X 3.2241,Y 44.034,Z 62,A 78.1618,B 24.837,C -2.9449,E1 25.0137,E2 -714.8222} C_DIS
LIN {X 5.4893,Y 43.809,Z 62,A 74.9442,B 24.8375,C -2.9405,E1 25.0227,E2 -711.5964} C_DIS
LIN {X 8.3723,Y 43.3501,Z 62,A 71.2861,B 24.8375,C -2.9412,E1 25.0327,E2 -707.9438} C_DIS
LIN {X 10.8186,Y 42.8056,Z 62,A 68.0297,B 24.8376,C -2.9394,E1 25.0416,E2 -704.6877} C_DIS
LIN {X 13.2223,Y 42.1251,Z 62,A 64.5745,B 24.8383,C -2.9338,E1 25.0508,E2 -701.2252} C_DIS
LIN {X 15.8055,Y 41.2256,Z 62,A 60.4623,B 24.8396,C -2.9219,E1 25.0616,E2 -697.0934} C_DIS
LIN {X 18.5418,Y 40.0692,Z 62,A 57.5991,B 24.8383,C -2.9332,E1 25.0689,E2 -694.2642} C_DIS
LIN {X 20.3322,Y 39.1918,Z 62,A 55.0247,B 24.8387,C -2.9302,E1 25.0753,E2 -691.6897} C_DIS
LIN {X 22.2484,Y 38.1366,Z 62,A 51.9267,B 24.8395,C -2.9221,E1 25.0828,E2 -688.5817} C_DIS
LIN {X 24.4709,Y 36.7497,Z 62,A 48.5592,B 24.8401,C -2.9175,E1 25.0907,E2 -685.2142} C_DIS
LIN {X 26.6192,Y 35.2245,Z 62,A 45.0675,B 24.8408,C -2.9105,E1 25.0986,E2 -681.7184} C_DIS
LIN {X 29.1283,Y 33.1796,Z 62,A 40.7233,B 24.8419,C -2.9002,E1 25.1079,E2 -677.3667} C_DIS
LIN {X 31.0894,Y 31.3494,Z 62,A 37.4748,B 24.8423,C -2.8971,E1 25.1144,E2 -674.1242} C_DIS
LIN {X 32.8264,Y 29.5256,Z 62,A 33.9812,B 24.8435,C -2.8862,E1 25.121,E2 -670.6201} C_DIS
LIN {X 34.9363,Y 26.996,Z 62,A 30.3263,B 24.8435,C -2.8869,E1 25.1274,E2 -666.9839} C_DIS
LIN {X 36.2533,Y 25.1997,Z 62,A 27.1257,B 24.8448,C -2.8745,E1 25.1326,E2 -663.7695} C_DIS
LIN {X 37.737,Y 22.9183,Z 62,A 23.8744,B 24.8452,C -2.8704,E1 25.1375,E2 -660.5248} C_DIS
LIN {X 38.8404,Y 20.9942,Z 62,A 20.965,B 24.8461,C -2.8623,E1 25.1415,E2 -657.6113} C_DIS
LIN {X 39.8568,Y 18.9943,Z 62,A 18.2849,B 24.8465,C -2.8584,E1 25.1448,E2 -654.9364} C_DIS
LIN {X 40.5731,Y 17.4131,Z 62,A 15.7096,B 24.8478,C -2.8464,E1 25.1477,E2 -652.3468} C_DIS
LIN {X 41.4504,Y 15.2052,Z 62,A 12.5095,B 24.8489,C -2.8356,E1 25.1509,E2 -649.1388} C_DIS
LIN {X 42.3292,Y 12.5525,Z 62,A 8.9766,B 24.8499,C -2.8266,E1 25.1538,E2 -645.6048} C_DIS
LIN {X 42.9128,Y 10.3838,Z 62,A 6.0588,B 24.8508,C -2.8178,E1 25.1558,E2 -642.6831} C_DIS
LIN {X 43.4702,Y 7.7252,Z 62,A 2.6246,B 24.8518,C -2.8088,E1 25.1577,E2 -639.2475} C_DIS
LIN {X 43.7826,Y 5.6935,Z 62,A -0.0842,B 24.8527,C -2.7998,E1 25.1587,E2 -636.5334} C_DIS
LIN {X 44.0519,Y 2.9599,Z 62,A -3.6128,B 24.8538,C -2.7894,E1 25.1596,E2 -633.0011} C_DIS
LIN {X 44.1458,Y 0.6978,Z 62,A -6.2924,B 24.8543,C -2.7848,E1 25.1598,E2 -630.3267} C_DIS
LIN {X 44.1258,Y -1.5023,Z 62,A -9.268,B 24.8555,C -2.7737,E1 25.1596,E2 -627.3425} C_DIS
LIN {X 44.0088,Y -3.5429,Z 62,A -11.9618,B 24.8564,C -2.7646,E1 25.1591,E2 -624.6432} C_DIS
LIN {X 43.7353,Y -6.0482,Z 62,A -15.2023,B 24.8575,C -2.7549,E1 25.158,E2 -621.3988} C_DIS
LIN {X 43.3398,Y -8.426,Z 62,A -18.2762,B 24.8584,C -2.7461,E1 25.1564,E2 -618.322} C_DIS
LIN {X 42.8109,Y -10.7979,Z 62,A -21.43,B 24.8594,C -2.7363,E1 25.1544,E2 -615.1633} C_DIS
LIN {X 42.2475,Y -12.8275,Z 62,A -23.8993,B 24.8598,C -2.7326,E1 25.1525,E2 -612.6995} C_DIS
LIN {X 41.6707,Y -14.5905,Z 62,A -26.6669,B 24.8612,C -2.7188,E1 25.15,E2 -609.9149} C_DIS
LIN {X 40.3471,Y -17.9301,Z 62,A -31.2092,B 24.8624,C -2.7071,E1 25.1451,E2 -605.3697} C_DIS
LIN {X 39.3277,Y -20.0665,Z 62,A -34.2243,B 24.8632,C -2.6991,E1 25.1414,E2 -602.352} C_DIS
LIN {X 38.1616,Y -22.2053,Z 62,A -37.2776,B 24.8639,C -2.6921,E1 25.1372,E2 -599.2978} C_DIS
LIN {X 36.7544,Y -24.4634,Z 62,A -40.8949,B 24.8652,C -2.6796,E1 25.1318,E2 -595.6693} C_DIS
LIN {X 35.5967,Y -26.119,Z 62,A -43.0716,B 24.8651,C -2.6804,E1 25.1282,E2 -593.5051} C_DIS
LIN {X 34.3669,Y -27.7174,Z 62,A -46.0197,B 24.8664,C -2.6678,E1 25.1231,E2 -590.5409} C_DIS
LIN {X 32.7551,Y -29.6053,Z 62,A -49.2528,B 24.8672,C -2.6595,E1 25.1171,E2 -587.3027} C_DIS
LIN {X 31.1819,Y -31.258,Z 62,A -52.2312,B 24.8679,C -2.6521,E1 25.1113,E2 -584.3195} C_DIS
LIN {X 29.1753,Y -33.1384,Z 62,A -55.7355,B 24.8686,C -2.6451,E1 25.1041,E2 -580.8128} C_DIS
LIN {X 27.5833,Y -34.4755,Z 62,A -58.4197,B 24.8692,C -2.6395,E1 25.0983,E2 -578.1254} C_DIS
LIN {X 25.6272,Y -35.9524,Z 62,A -61.5453,B 24.8697,C -2.634,E1 25.0912,E2 -574.9979} C_DIS
LIN {X 23.5648,Y -37.3372,Z 62,A -64.8241,B 24.8704,C -2.6269,E1 25.0835,E2 -571.7131} C_DIS
LIN {X 21.3043,Y -38.6719,Z 62,A -68.1853,B 24.8709,C -2.6217,E1 25.0754,E2 -568.3495} C_DIS
LIN {X 19.0475,Y -39.8312,Z 62,A -71.523,B 24.8715,C -2.6157,E1 25.067,E2 -565.0066} C_DIS
LIN {X 17.2106,Y -40.6587,Z 62,A -74.0927,B 24.8718,C -2.6126,E1 25.0604,E2 -562.4358} C_DIS
LIN {X 14.2369,Y -41.793,Z 62,A -77.7084,B 24.8715,C -2.6156,E1 25.051,E2 -558.8348} C_DIS
LIN {X 12.4877,Y -42.3484,Z 62,A -80.6102,B 24.8726,C -2.6045,E1 25.0432,E2 -555.9119} C_DIS
LIN {X 10.2313,Y -42.95,Z 62,A -83.4589,B 24.8726,C -2.6044,E1 25.0355,E2 -553.0671} C_DIS
LIN {X 8.0124,Y -43.4185,Z 62,A -86.4233,B 24.8729,C -2.6016,E1 25.0274,E2 -550.0997} C_DIS
LIN {X 5.8972,Y -43.7562,Z 62,A -89.1768,B 24.8731,C -2.6001,E1 25.0198,E2 -547.3451} C_DIS
LIN {X 3.7717,Y -43.9905,Z 62,A -91.9969,B 24.8733,C -2.5979,E1 25.0119,E2 -544.5216} C_DIS
LIN {X 1.6561,Y -44.1208,Z 62,A -94.822,B 24.8735,C -2.5957,E1 25.004,E2 -541.6923} C_DIS
LIN {X 0.2247,Y -44.1474,Z 62,A -96.7457,B 24.8736,C -2.5943,E1 24.9986,E2 -539.7654} C_DIS
Enddeposition()
LIN {X 0.2247,Y -44.1474,Z 62,A -96.7457,B 24.8736,C -2.5943,E1 24.9986,E2 -539.7654} C_DIS
Startdeposition()
$VEL.CP = VEL_PRINT
LIN {X 0.5538,Y -43.1685,Z 62,A -94.8369,B 24.8698,C -2.6337,E1 25.0042,E2 -541.7676} C_DIS
LIN {X 3.2483,Y -43.0496,Z 62,A -91.1094,B 24.8694,C -2.6374,E1 25.0146,E2 -545.5025} C_DIS
LIN {X 5.71,Y -42.7926,Z 62,A -88.31,B 24.8699,C -2.6318,E1 25.0224,E2 -548.2865} C_DIS
LIN {X 7.3625,Y -42.5389,Z 62,A -85.8174,B 24.8694,C -2.6377,E1 25.0293,E2 -550.7907} C_DIS
LIN {X 9.4175,Y -42.1315,Z 62,A -82.6035,B 24.8684,C -2.647,E1 25.0381,E2 -554.0225} C_DIS
LIN {X 12.1349,Y -41.4312,Z 62,A -78.745,B 24.8678,C -2.6531,E1 25.0485,E2 -557.8893} C_DIS
LIN {X 14.4098,Y -40.6959,Z 62,A -75.9472,B 24.868,C -2.6509,E1 25.0559,E2 -560.6763} C_DIS
LIN {X 16.8357,Y -39.7536,Z 62,A -72.8015,B 24.868,C -2.6507,E1 25.064,E2 -563.8143} C_DIS
LIN {X 19.0885,Y -38.7217,Z 62,A -69.5472,B 24.8676,C -2.6552,E1 25.0722,E2 -567.0709} C_DIS
LIN {X 20.6538,Y -37.9104,Z 62,A -66.6299,B 24.8663,C -2.6687,E1 25.0794,E2 -570.012} C_DIS
LIN {X 23.195,Y -36.4115,Z 62,A -63.0541,B 24.8661,C -2.6702,E1 25.0879,E2 -573.58} C_DIS
LIN {X 25.0449,Y -35.1644,Z 62,A -60.0395,B 24.8654,C -2.677,E1 25.0949,E2 -576.6002} C_DIS
LIN {X 26.9397,Y -33.7355,Z 62,A -56.8241,B 24.8646,C -2.6847,E1 25.102,E2 -579.8222} C_DIS
LIN {X 28.8704,Y -32.0981,Z 62,A -53.6963,B 24.8643,C -2.6882,E1 25.1085,E2 -582.946} C_DIS
LIN {X 30.5952,Y -30.4588,Z 62,A -50.4335,B 24.8634,C -2.6975,E1 25.1151,E2 -586.217} C_DIS
LIN {X 32.2474,Y -28.7037,Z 62,A -47.3532,B 24.8628,C -2.7033,E1 25.1209,E2 -589.2976} C_DIS
LIN {X 33.6707,Y -27.0205,Z 62,A -44.8022,B 24.8627,C -2.7042,E1 25.1254,E2 -591.839} C_DIS
LIN {X 34.9233,Y -25.3804,Z 62,A -41.5469,B 24.861,C -2.7206,E1 25.1309,E2 -595.1174} C_DIS
LIN {X 36.1541,Y -23.5945,Z 62,A -39.0259,B 24.8608,C -2.7221,E1 25.1348,E2 -597.6295} C_DIS
LIN {X 37.4338,Y -21.5056,Z 62,A -35.2035,B 24.8588,C -2.7414,E1 25.1403,E2 -601.478} C_DIS
LIN {X 38.7575,Y -19.0175,Z 62,A -31.968,B 24.8587,C -2.7432,E1 25.1443,E2 -604.7005} C_DIS
LIN {X 39.635,Y -17.1134,Z 62,A -29.2001,B 24.8578,C -2.7512,E1 25.1475,E2 -607.4722} C_DIS
LIN {X 40.3694,Y -15.3001,Z 62,A -26.398,B 24.8566,C -2.7627,E1 25.1503,E2 -610.286} C_DIS
LIN {X 41.1441,Y -13.0766,Z 62,A -22.977,B 24.8551,C -2.7775,E1 25.1533,E2 -613.7228} C_DIS
LIN {X 42.1051,Y -9.5382,Z 62,A -18.5082,B 24.8543,C -2.7854,E1 25.1564,E2 -618.1844} C_DIS
LIN {X 42.5881,Y -7.0738,Z 62,A -15.2351,B 24.8533,C -2.7947,E1 25.158,E2 -621.4604} C_DIS
LIN {X 42.8853,Y -4.9638,Z 62,A -12.8054,B 24.8531,C -2.7964,E1 25.1589,E2 -623.8798} C_DIS
LIN {X 43.0666,Y -3.0103,Z 62,A -9.923,B 24.8517,C -2.8096,E1 25.1595,E2 -626.7763} C_DIS
LIN {X 43.1565,Y -1.1504,Z 62,A -7.2779,B 24.8506,C -2.8205,E1 25.1598,E2 -629.4315} C_DIS
LIN {X 43.1443,Y 1.5511,Z 62,A -3.944,B 24.8498,C -2.8272,E1 25.1596,E2 -632.7613} C_DIS
LIN {X 43.0157,Y 3.6722,Z 62,A -1.1244,B 24.8489,C -2.836,E1 25.159,E2 -635.585} C_DIS
LIN {X 42.7073,Y 6.3188,Z 62,A 2.7482,B 24.8471,C -2.8529,E1 25.1576,E2 -639.4748} C_DIS
LIN {X 42.2272,Y 8.983,Z 62,A 5.9329,B 24.8467,C -2.8565,E1 25.1559,E2 -642.6494} C_DIS
LIN {X 41.7456,Y 11.007,Z 62,A 8.6719,B 24.8459,C -2.8644,E1 25.154,E2 -645.3912} C_DIS
LIN {X 41.1668,Y 13.005,Z 62,A 11.6699,B 24.8445,C -2.8767,E1 25.1515,E2 -648.4014} C_DIS
LIN {X 40.1108,Y 15.9669,Z 62,A 15.6937,B 24.8435,C -2.886,E1 25.1476,E2 -652.4247} C_DIS
LIN {X 38.5379,Y 19.459,Z 62,A 20.5211,B 24.8425,C -2.8955,E1 25.1419,E2 -657.2485} C_DIS
LIN {X 37.6699,Y 21.0894,Z 62,A 23.567,B 24.8406,C -2.9124,E1 25.1378,E2 -660.3185} C_DIS
LIN {X 36.0816,Y 23.7045,Z 62,A 27.0869,B 24.8406,C -2.9133,E1 25.1326,E2 -663.8228} C_DIS
LIN {X 34.8997,Y 25.4126,Z 62,A 29.8128,B 24.8398,C -2.9195,E1 25.1281,E2 -666.5501} C_DIS
LIN {X 32.7927,Y 28.0786,Z 62,A 34.2176,B 24.8389,C -2.9281,E1 25.1204,E2 -670.9548} C_DIS
LIN {X 31.6923,Y 29.3152,Z 62,A 36.6636,B 24.8379,C -2.9371,E1 25.1158,E2 -673.4114} C_DIS
LIN {X 29.7253,Y 31.3086,Z 62,A 41.244,B 24.8354,C -2.9593,E1 25.1065,E2 -678.0252} C_DIS
LIN {X 27.067,Y 33.633,Z 62,A 44.9567,B 24.8363,C -2.9517,E1 25.0986,E2 -681.7056} C_DIS
LIN {X 25.2071,Y 35.0487,Z 62,A 48.1307,B 24.8356,C -2.9581,E1 25.0915,E2 -684.8835} C_DIS
LIN {X 23.0773,Y 36.4866,Z 62,A 51.553,B 24.8349,C -2.9636,E1 25.0835,E2 -688.3076} C_DIS
LIN {X 21.3925,Y 37.4988,Z 62,A 54.376,B 24.8341,C -2.9707,E1 25.0766,E2 -691.139} C_DIS
LIN {X 18.6887,Y 38.9168,Z 62,A 57.9628,B 24.8344,C -2.9683,E1 25.0677,E2 -694.7103} C_DIS
LIN {X 16.0359,Y 40.0836,Z 62,A 62.1541,B 24.8334,C -2.9777,E1 25.0569,E2 -698.914} C_DIS
LIN {X 13.2505,Y 41.0878,Z 62,A 66.2902,B 24.8326,C -2.9841,E1 25.046,E2 -703.0574} C_DIS
LIN {X 10.3647,Y 41.9091,Z 62,A 69.894,B 24.833,C -2.9807,E1 25.0363,E2 -706.6475} C_DIS
LIN {X 8.3709,Y 42.3527,Z 62,A 72.606,B 24.8329,C -2.982,E1 25.0289,E2 -709.3591} C_DIS
LIN {X 6.0804,Y 42.7412,Z 62,A 75.4735,B 24.8331,C -2.9796,E1 25.021,E2 -712.2183} C_DIS
LIN {X 3.661,Y 43.0166,Z 62,A 78.8371,B 24.8329,C -2.982,E1 25.0116,E2 -715.5852} C_DIS
LIN {X 1.2569,Y 43.1533,Z 62,A 82.0248,B 24.8329,C -2.9817,E1 25.0027,E2 -718.7713} C_DIS
LIN {X -1.8775,Y 43.1307,Z 62,A 86.419,B 24.8327,C -2.9839,E1 24.9904,E2 -723.1713} C_DIS
LIN {X -4.3229,Y 42.9549,Z 62,A 89.3239,B 24.8334,C -2.9775,E1 24.9824,E2 -726.0622} C_DIS
LIN {X -6.2162,Y 42.7215,Z 62,A 92.3251,B 24.8328,C -2.9825,E1 24.9741,E2 -729.0777} C_DIS
LIN {X -9.06,Y 42.2104,Z 62,A 95.4714,B 24.8342,C -2.9699,E1 24.9655,E2 -732.1976} C_DIS
LIN {X -11.5301,Y 41.604,Z 62,A 99.739,B 24.8332,C -2.9788,E1 24.9539,E2 -736.4926} C_DIS
LIN {X -14.0785,Y 40.8119,Z 62,A 102.543,B 24.8348,C -2.9647,E1 24.9466,E2 -739.2682} C_DIS
LIN {X -16.7156,Y 39.8042,Z 62,A 106.4886,B 24.8351,C -2.9624,E1 24.9363,E2 -743.2168} C_DIS
LIN {X -18.3788,Y 39.0645,Z 62,A 108.8793,B 24.8355,C -2.9585,E1 24.9302,E2 -745.6041} C_DIS
LIN {X -20.7212,Y 37.874,Z 62,A 112.0502,B 24.8366,C -2.9487,E1 24.9224,E2 -748.7603} C_DIS
LIN {X -22.3055,Y 36.963,Z 62,A 114.7882,B 24.8366,C -2.9485,E1 24.9158,E2 -751.5061} C_DIS
LIN {X -24.4768,Y 35.5626,Z 62,A 118.6485,B 24.8367,C -2.9475,E1 24.9068,E2 -755.3767} C_DIS
LIN {X -26.3498,Y 34.1975,Z 62,A 121.4408,B 24.8378,C -2.9376,E1 24.9006,E2 -758.1555} C_DIS
LIN {X -27.843,Y 32.9933,Z 62,A 124.6111,B 24.8376,C -2.9399,E1 24.8938,E2 -761.3436} C_DIS
LIN {X -30.7202,Y 30.3324,Z 62,A 129.5686,B 24.8392,C -2.9248,E1 24.8839,E2 -766.2856} C_DIS
LIN {X -33.2367,Y 27.5514,Z 62,A 134.2664,B 24.841,C -2.909,E1 24.8753,E2 -770.9668} C_DIS
LIN {X -35.1946,Y 25.0026,Z 62,A 138.3775,B 24.8424,C -2.896,E1 24.8685,E2 -775.0664} C_DIS
LIN {X -36.9462,Y 22.3332,Z 62,A 142.7731,B 24.8435,C -2.8862,E1 24.8619,E2 -779.461} C_DIS
LIN {X -37.7874,Y 20.8789,Z 62,A 145.3173,B 24.8438,C -2.8836,E1 24.8584,E2 -782.0123} C_DIS
LIN {X -39.0298,Y 18.4532,Z 62,A 148.5873,B 24.8453,C -2.869,E1 24.8544,E2 -785.265} C_DIS
LIN {X -39.7383,Y 16.872,Z 62,A 150.9021,B 24.8461,C -2.8624,E1 24.8518,E2 -787.5768} C_DIS
LIN {X -40.5761,Y 14.7433,Z 62,A 154.0861,B 24.8469,C -2.855,E1 24.8487,E2 -790.761} C_DIS
LIN {X -41.2607,Y 12.7021,Z 62,A 156.9098,B 24.8478,C -2.846,E1 24.8463,E2 -793.5793} C_DIS
LIN {X -41.8918,Y 10.4339,Z 62,A 160.038,B 24.8489,C -2.8364,E1 24.844,E2 -796.7027} C_DIS
LIN {X -42.402,Y 8.1151,Z 62,A 163.2233,B 24.8499,C -2.827,E1 24.8422,E2 -799.8844} C_DIS
LIN {X -42.8263,Y 5.4496,Z 62,A 167.0557,B 24.8507,C -2.8187,E1 24.8407,E2 -803.7197} C_DIS
LIN {X -43.0515,Y 3.2221,Z 62,A 169.6825,B 24.8522,C -2.8054,E1 24.8401,E2 -806.3304} C_DIS
LIN {X -43.1565,Y 1.1532,Z 62,A 172.6629,B 24.8528,C -2.7994,E1 24.8398,E2 -809.3145} C_DIS
LIN {X -43.1645,Y -0.7777,Z 62,A 175.6282,B 24.8531,C -2.7961,E1 24.8399,E2 -812.2897} C_DIS
LIN {X -42.9646,Y -4.2241,Z 62,A 179.8432,B 24.8551,C -2.7776,E1 24.8408,E2 -816.4857} C_DIS
LIN {X -42.473,Y -7.7354,Z 62,A -175.3959,B 24.8565,C -2.7638,E1 24.8428,E2 -821.242} C_DIS
LIN {X -42.0692,Y -9.6934,Z 62,A -172.8948,B 24.8575,C -2.754,E1 24.8443,E2 -823.7345} C_DIS
LIN {X -41.4394,Y -12.1074,Z 62,A -169.2286,B 24.8581,C -2.7484,E1 24.8471,E2 -827.4085} C_DIS
LIN {X -40.556,Y -14.7983,Z 62,A -165.686,B 24.8595,C -2.735,E1 24.8503,E2 -830.939} C_DIS
LIN {X -39.7167,Y -16.9231,Z 62,A -163.0702,B 24.8609,C -2.7215,E1 24.853,E2 -833.5371} C_DIS
LIN {X -38.9601,Y -18.5985,Z 62,A -160.2244,B 24.8611,C -2.7196,E1 24.8564,E2 -836.394} C_DIS
LIN {X -37.9405,Y -20.5986,Z 62,A -157.1118,B 24.8617,C -2.7133,E1 24.8604,E2 -839.508} C_DIS
LIN {X -36.6995,Y -22.7366,Z 62,A -153.7473,B 24.8625,C -2.7058,E1 24.8653,E2 -842.8721} C_DIS
LIN {X -35.3326,Y -24.8078,Z 62,A -150.5743,B 24.8635,C -2.6962,E1 24.8702,E2 -846.0379} C_DIS
LIN {X -34.0969,Y -26.4803,Z 62,A -147.5652,B 24.8638,C -2.6928,E1 24.8753,E2 -849.0532} C_DIS
LIN {X -32.3286,Y -28.613,Z 62,A -143.9701,B 24.8648,C -2.6836,E1 24.8819,E2 -852.6426} C_DIS
LIN {X -30.5606,Y -30.4939,Z 62,A -141.0785,B 24.8662,C -2.6696,E1 24.8874,E2 -855.5133} C_DIS
LIN {X -29.2707,Y -31.7336,Z 62,A -137.8118,B 24.8655,C -2.6763,E1 24.8941,E2 -858.8095} C_DIS
LIN {X -27.0563,Y -33.6417,Z 62,A -134.4218,B 24.8669,C -2.6628,E1 24.9014,E2 -862.1802} C_DIS
LIN {X -25.1713,Y -35.0743,Z 62,A -131.5841,B 24.8678,C -2.6535,E1 24.9077,E2 -865.0058} C_DIS
LIN {X -23.0177,Y -36.5239,Z 62,A -127.5593,B 24.8675,C -2.6559,E1 24.9171,E2 -869.0496} C_DIS
LIN {X -20.7039,Y -37.8833,Z 62,A -124.7268,B 24.869,C -2.6413,E1 24.9239,E2 -871.8554} C_DIS
LIN {X -18.9771,Y -38.7775,Z 62,A -121.3252,B 24.8682,C -2.6493,E1 24.9325,E2 -875.2853} C_DIS
LIN {X -17.0989,Y -39.6414,Z 62,A -118.8704,B 24.8689,C -2.6424,E1 24.9387,E2 -877.7295} C_DIS
LIN {X -14.6328,Y -40.6164,Z 62,A -115.261,B 24.8691,C -2.6405,E1 24.9482,E2 -881.342} C_DIS
LIN {X -12.2481,Y -41.3977,Z 62,A -112.2143,B 24.8697,C -2.6341,E1 24.9562,E2 -884.3787} C_DIS
LIN {X -9.4259,Y -42.13,Z 62,A -107.6032,B 24.8689,C -2.6428,E1 24.9688,E2 -889.0168} C_DIS
LIN {X -6.2993,Y -42.7099,Z 62,A -103.7779,B 24.8696,C -2.6357,E1 24.9793,E2 -892.829} C_DIS
LIN {X -3.8376,Y -43.0008,Z 62,A -100.577,B 24.8697,C -2.6341,E1 24.9882,E2 -896.0278} C_DIS
LIN {X -1.4573,Y -43.1471,Z 62,A -97.4985,B 24.8698,C -2.633,E1 24.9968,E2 -899.1046} C_DIS
LIN {X 0.2235,Y -43.1689,Z 62,A -96.1407,B 24.8711,C -2.6204,E1 25.0005,E2 -900.4324} C_DIS
Enddeposition()
LIN {X 0.2235,Y -43.1689,Z 62,A -96.1407,B 24.8711,C -2.6204,E1 25.0005,E2 -900.4324} C_DIS
Startdeposition()
$VEL.CP = VEL_PRINT
LIN {X -1.0904,Y -42.1779,Z 62,A -98.9049,B 24.8708,C -2.623,E1 24.9928,E2 -897.6742} C_DIS
LIN {X -3.2026,Y -42.0705,Z 62,A -101.4005,B 24.8703,C -2.6283,E1 24.9859,E2 -895.1902} C_DIS
LIN {X -5.6023,Y -41.8187,Z 62,A -104.9545,B 24.8706,C -2.6249,E1 24.976,E2 -891.6257} C_DIS
LIN {X -7.9617,Y -41.4339,Z 62,A -107.5894,B 24.8697,C -2.6345,E1 24.9688,E2 -889.0108} C_DIS
LIN {X -10.009,Y -40.9875,Z 62,A -111.1214,B 24.8705,C -2.6265,E1 24.9591,E2 -885.4551} C_DIS
LIN {X -12.8572,Y -40.1854,Z 62,A -114.8378,B 24.8698,C -2.6333,E1 24.9492,E2 -881.7487} C_DIS
LIN {X -15.2278,Y -39.3486,Z 62,A -118.2459,B 24.8695,C -2.6363,E1 24.9403,E2 -878.3409} C_DIS
LIN {X -17.3785,Y -38.4467,Z 62,A -121.3606,B 24.8691,C -2.6403,E1 24.9323,E2 -875.2284} C_DIS
LIN {X -19.6411,Y -37.3414,Z 62,A -124.8268,B 24.8687,C -2.6439,E1 24.9237,E2 -871.7613} C_DIS
LIN {X -21.8754,Y -36.078,Z 62,A -127.9674,B 24.8678,C -2.6531,E1 24.9161,E2 -868.6334} C_DIS
LIN {X -23.6214,Y -34.9598,Z 62,A -131.4821,B 24.8683,C -2.6486,E1 24.9079,E2 -865.0964} C_DIS
LIN {X -25.3149,Y -33.7537,Z 62,A -134.0048,B 24.8674,C -2.6571,E1 24.9023,E2 -862.585} C_DIS
LIN {X -27.6499,Y -31.8687,Z 62,A -138.0635,B 24.8667,C -2.6648,E1 24.8936,E2 -858.5291} C_DIS
LIN {X -29.2286,Y -30.4271,Z 62,A -141.0083,B 24.8661,C -2.67,E1 24.8876,E2 -855.5848} C_DIS
LIN {X -30.9954,Y -28.6262,Z 62,A -144.4701,B 24.8654,C -2.6768,E1 24.8809,E2 -852.1243} C_DIS
LIN {X -32.8025,Y -26.535,Z 62,A -147.9606,B 24.8643,C -2.6884,E1 24.8746,E2 -848.6455} C_DIS
LIN {X -34.2164,Y -24.6853,Z 62,A -151.7308,B 24.8643,C -2.6889,E1 24.8683,E2 -844.8581} C_DIS
LIN {X -35.6707,Y -22.5344,Z 62,A -155.3457,B 24.8634,C -2.6967,E1 24.8629,E2 -841.2437} C_DIS
LIN {X -37.2253,Y -19.8613,Z 62,A -158.8987,B 24.8616,C -2.7151,E1 24.858,E2 -837.7161} C_DIS
LIN {X -37.9178,Y -18.5051,Z 62,A -161.1386,B 24.8612,C -2.7187,E1 24.8552,E2 -835.4728} C_DIS
LIN {X -38.8285,Y -16.5083,Z 62,A -163.8556,B 24.86,C -2.73,E1 24.8522,E2 -832.7678} C_DIS
LIN {X -39.4878,Y -14.8619,Z 62,A -166.8386,B 24.86,C -2.7304,E1 24.8492,E2 -829.769} C_DIS
LIN {X -40.2123,Y -12.7723,Z 62,A -169.8907,B 24.8591,C -2.7386,E1 24.8465,E2 -826.7191} C_DIS
LIN {X -41.0634,Y -9.6937,Z 62,A -173.8457,B 24.8574,C -2.7557,E1 24.8437,E2 -822.782} C_DIS
LIN {X -41.6337,Y -6.8416,Z 62,A -178.6769,B 24.8571,C -2.7581,E1 24.8413,E2 -817.9279} C_DIS
LIN {X -42.1023,Y -2.7497,Z 62,A 175.945,B 24.8551,C -2.7778,E1 24.8399,E2 -812.5647} C_DIS
LIN {X -42.1914,Y 0.2062,Z 62,A 171.8104,B 24.8539,C -2.7891,E1 24.8399,E2 -808.4321} C_DIS
LIN {X -42.0233,Y 3.7695,Z 62,A 167.4663,B 24.8517,C -2.8097,E1 24.8406,E2 -804.1112} C_DIS
LIN {X -41.7582,Y 6.0312,Z 62,A 164.4502,B 24.8506,C -2.8202,E1 24.8417,E2 -801.1022} C_DIS
LIN {X -41.4434,Y 7.912,Z 62,A 161.2223,B 24.8505,C -2.8214,E1 24.8433,E2 -797.858} C_DIS
LIN {X -40.5134,Y 11.7844,Z 62,A 155.852,B 24.8486,C -2.8384,E1 24.8471,E2 -792.4973} C_DIS
LIN {X -39.4968,Y 14.8382,Z 62,A 152.3102,B 24.8462,C -2.8607,E1 24.8504,E2 -788.9886} C_DIS
LIN {X -38.8671,Y 16.4168,Z 62,A 149.6499,B 24.8459,C -2.8637,E1 24.8532,E2 -786.3207} C_DIS
LIN {X -37.9982,Y 18.3383,Z 62,A 146.965,B 24.8448,C -2.874,E1 24.8563,E2 -783.6459} C_DIS
LIN {X -37.1756,Y 19.9523,Z 62,A 143.8606,B 24.8448,C -2.874,E1 24.8604,E2 -780.5248} C_DIS
LIN {X -35.6018,Y 22.6424,Z 62,A 140.0965,B 24.843,C -2.8909,E1 24.8658,E2 -776.7819} C_DIS
LIN {X -34.6538,Y 24.0681,Z 62,A 137.6307,B 24.8425,C -2.8956,E1 24.8697,E2 -774.3151} C_DIS
LIN {X -33.3498,Y 25.8449,Z 62,A 134.7044,B 24.8415,C -2.9042,E1 24.8746,E2 -771.3954} C_DIS
LIN {X -32.2288,Y 27.2303,Z 62,A 132.3621,B 24.8407,C -2.9112,E1 24.8787,E2 -769.059} C_DIS
LIN {X -30.8683,Y 28.7635,Z 62,A 129.2648,B 24.8404,C -2.9144,E1 24.8845,E2 -765.9556} C_DIS
LIN {X -29.1201,Y 30.5323,Z 62,A 125.7593,B 24.8397,C -2.9208,E1 24.8915,E2 -762.4507} C_DIS
LIN {X -27.5908,Y 31.9208,Z 62,A 123.2995,B 24.8386,C -2.9311,E1 24.8966,E2 -760.0057} C_DIS
LIN {X -26.3111,Y 32.9836,Z 62,A 120.4765,B 24.8388,C -2.9292,E1 24.9028,E2 -757.1677} C_DIS
LIN {X -23.6646,Y 34.9301,Z 62,A 116.6998,B 24.8369,C -2.9462,E1 24.9113,E2 -753.4185} C_DIS
LIN {X -22.3422,Y 35.7908,Z 62,A 114.2627,B 24.8369,C -2.9466,E1 24.9171,E2 -750.9745} C_DIS
LIN {X -20.0031,Y 37.1484,Z 62,A 110.6253,B 24.8361,C -2.9533,E1 24.9259,E2 -747.3425} C_DIS
LIN {X -17.6727,Y 38.3125,Z 62,A 107.0255,B 24.8356,C -2.958,E1 24.9349,E2 -743.7445} C_DIS
LIN {X -15.0185,Y 39.4285,Z 62,A 102.9853,B 24.8352,C -2.9617,E1 24.9454,E2 -739.7041} C_DIS
LIN {X -12.6787,Y 40.2423,Z 62,A 99.8366,B 24.8344,C -2.9684,E1 24.9537,E2 -736.5654} C_DIS
LIN {X -10.9537,Y 40.7449,Z 62,A 97.1055,B 24.8345,C -2.9671,E1 24.9611,E2 -733.8272} C_DIS
LIN {X -8.2509,Y 41.3779,Z 62,A 93.3405,B 24.8342,C -2.9704,E1 24.9713,E2 -730.0652} C_DIS
LIN {X -5.5334,Y 41.8276,Z 62,A 89.554,B 24.834,C -2.9722,E1 24.9818,E2 -726.28} C_DIS
LIN {X -3.2334,Y 42.068,Z 62,A 86.6834,B 24.8334,C -2.9774,E1 24.9898,E2 -723.4201} C_DIS
LIN {X -1.2057,Y 42.1747,Z 62,A 83.7403,B 24.8336,C -2.9757,E1 24.998,E2 -720.4725} C_DIS
LIN {X 1.0967,Y 42.1781,Z 62,A 80.2358,B 24.8341,C -2.9709,E1 25.0078,E2 -716.9572} C_DIS
LIN {X 4.285,Y 41.9739,Z 62,A 76.467,B 24.8332,C -2.9787,E1 25.0182,E2 -713.2087} C_DIS
LIN {X 6.8959,Y 41.6246,Z 62,A 72.3238,B 24.8343,C -2.9697,E1 25.0297,E2 -709.0478} C_DIS
LIN {X 9.6606,Y 41.0713,Z 62,A 68.8489,B 24.8339,C -2.9729,E1 25.0392,E2 -705.5853} C_DIS
LIN {X 12.1849,Y 40.3946,Z 62,A 65.2587,B 24.8342,C -2.9699,E1 25.0488,E2 -701.994} C_DIS
LIN {X 14.4207,Y 39.651,Z 62,A 62.1743,B 24.8343,C -2.9689,E1 25.0569,E2 -698.9135} C_DIS
LIN {X 16.7424,Y 38.7281,Z 62,A 59.0061,B 24.8343,C -2.9689,E1 25.0651,E2 -695.7524} C_DIS
LIN {X 18.7824,Y 37.7807,Z 62,A 56.0976,B 24.8345,C -2.9676,E1 25.0724,E2 -692.8483} C_DIS
LIN {X 20.5125,Y 36.87,Z 62,A 52.9906,B 24.8357,C -2.9571,E1 25.0801,E2 -689.7254} C_DIS
LIN {X 22.4312,Y 35.7352,Z 62,A 50.0784,B 24.836,C -2.9544,E1 25.087,E2 -686.8161} C_DIS
LIN {X 24.4783,Y 34.3653,Z 62,A 46.6077,B 24.8368,C -2.9471,E1 25.095,E2 -683.3398} C_DIS
LIN {X 26.3653,Y 32.9407,Z 62,A 43.7712,B 24.8368,C -2.9473,E1 25.1012,E2 -680.5142} C_DIS
LIN {X 27.5193,Y 31.9819,Z 62,A 40.969,B 24.8385,C -2.9313,E1 25.1072,E2 -677.6851} C_DIS
LIN {X 29.6471,Y 30.0201,Z 62,A 37.5577,B 24.8385,C -2.9317,E1 25.1141,E2 -674.2887} C_DIS
LIN {X 31.4993,Y 28.0705,Z 62,A 34.1781,B 24.8389,C -2.9282,E1 25.1205,E2 -670.9157} C_DIS
LIN {X 32.6034,Y 26.7801,Z 62,A 31.3667,B 24.8404,C -2.9147,E1 25.1255,E2 -668.0852} C_DIS
LIN {X 34.3384,Y 24.5159,Z 62,A 27.8059,B 24.8408,C -2.9106,E1 25.1314,E2 -664.5317} C_DIS
LIN {X 35.6636,Y 22.5458,Z 62,A 24.6531,B 24.8416,C -2.9036,E1 25.1362,E2 -661.3783} C_DIS
LIN {X 36.7355,Y 20.7532,Z 62,A 21.606,B 24.8428,C -2.8927,E1 25.1405,E2 -658.3211} C_DIS
LIN {X 37.7747,Y 18.7944,Z 62,A 18.5345,B 24.8438,C -2.8836,E1 25.1444,E2 -655.2442} C_DIS
LIN {X 39.0609,Y 15.95,Z 62,A 14.8369,B 24.8441,C -2.8809,E1 25.1485,E2 -651.5605} C_DIS
LIN {X 39.9104,Y 13.6882,Z 62,A 11.0426,B 24.846,C -2.8627,E1 25.1521,E2 -647.7444} C_DIS
LIN {X 40.6728,Y 11.2217,Z 62,A 7.8136,B 24.8466,C -2.8571,E1 25.1546,E2 -644.5206} C_DIS
LIN {X 41.2518,Y 8.8579,Z 62,A 4.219,B 24.8482,C -2.8422,E1 25.1569,E2 -640.9116} C_DIS
LIN {X 41.7394,Y 6.1671,Z 62,A 0.9065,B 24.8487,C -2.8377,E1 25.1584,E2 -637.608} C_DIS
LIN {X 42.0211,Y 3.7927,Z 62,A -2.0749,B 24.8493,C -2.8322,E1 25.1593,E2 -634.6313} C_DIS
LIN {X 42.156,Y 1.7408,Z 62,A -5.0987,B 24.8507,C -2.8195,E1 25.1597,E2 -631.5953} C_DIS
LIN {X 42.1763,Y -1.1564,Z 62,A -9.0259,B 24.852,C -2.8073,E1 25.1597,E2 -627.6626} C_DIS
LIN {X 42.0811,Y -3.0628,Z 62,A -11.358,B 24.8523,C -2.8037,E1 25.1592,E2 -625.3357} C_DIS
LIN {X 41.9003,Y -4.9523,Z 62,A -14.2065,B 24.8537,C -2.7909,E1 25.1584,E2 -622.4738} C_DIS
LIN {X 41.6215,Y -6.9143,Z 62,A -16.8628,B 24.8545,C -2.7831,E1 25.1572,E2 -619.8146} C_DIS
LIN {X 41.0624,Y -9.6943,Z 62,A -20.4866,B 24.8554,C -2.775,E1 25.1551,E2 -616.1929} C_DIS
LIN {X 40.4814,Y -11.891,Z 62,A -23.9142,B 24.857,C -2.7596,E1 25.1525,E2 -612.7485} C_DIS
LIN {X 39.9056,Y -13.7022,Z 62,A -26.4532,B 24.8577,C -2.7524,E1 25.1503,E2 -610.2069} C_DIS
LIN {X 38.9891,Y -16.1263,Z 62,A -29.7646,B 24.8584,C -2.7455,E1 25.1469,E2 -606.8973} C_DIS
LIN {X 38.0119,Y -18.3098,Z 62,A -32.6043,B 24.8587,C -2.743,E1 25.1436,E2 -604.0671} C_DIS
LIN {X 37.4005,Y -19.5276,Z 62,A -35.1482,B 24.8605,C -2.7257,E1 25.1403,E2 -601.4959} C_DIS
LIN {X 35.7199,Y -22.4557,Z 62,A -38.9087,B 24.8603,C -2.7269,E1 25.135,E2 -597.7574} C_DIS
LIN {X 34.1988,Y -24.7116,Z 62,A -43.7306,B 24.8633,C -2.6979,E1 25.1272,E2 -592.8904} C_DIS
LIN {X 32.1109,Y -27.3687,Z 62,A -47.6541,B 24.8633,C -2.6972,E1 25.1203,E2 -588.9836} C_DIS
LIN {X 29.6124,Y -30.0544,Z 62,A -52.2634,B 24.864,C -2.6913,E1 25.1114,E2 -584.3803} C_DIS
LIN {X 28.564,Y -31.0525,Z 62,A -54.9197,B 24.8656,C -2.6754,E1 25.1059,E2 -581.6972} C_DIS
LIN {X 25.5417,Y -33.5833,Z 62,A -59.8932,B 24.8661,C -2.6701,E1 25.0952,E2 -576.7299} C_DIS
LIN {X 23.5761,Y -34.9904,Z 62,A -63.8598,B 24.8679,C -2.6527,E1 25.086,E2 -572.7354} C_DIS
LIN {X 20.8459,Y -36.683,Z 62,A -67.8743,B 24.8681,C -2.6504,E1 25.0763,E2 -568.7278} C_DIS
LIN {X 17.8245,Y -38.2419,Z 62,A -72.0033,B 24.8681,C -2.6508,E1 25.066,E2 -564.6107} C_DIS
LIN {X 16.1354,Y -38.9848,Z 62,A -74.5708,B 24.8685,C -2.6462,E1 25.0594,E2 -562.0384} C_DIS
LIN {X 14.1123,Y -39.7621,Z 62,A -77.5654,B 24.869,C -2.6416,E1 25.0515,E2 -559.0391} C_DIS
LIN {X 11.322,Y -40.6448,Z 62,A -81.8154,B 24.8698,C -2.6329,E1 25.0401,E2 -554.776} C_DIS
LIN {X 8.5943,Y -41.3075,Z 62,A -85.3407,B 24.8698,C -2.6338,E1 25.0306,E2 -551.2575} C_DIS
LIN {X 5.8756,Y -41.7808,Z 62,A -89.0729,B 24.87,C -2.6313,E1 25.0203,E2 -547.5231} C_DIS
LIN {X 2.9966,Y -42.0856,Z 62,A -93.2604,B 24.8706,C -2.6256,E1 25.0086,E2 -543.3244} C_DIS
LIN {X 0.488,Y -42.1896,Z 62,A -96.6446,B 24.8706,C -2.6249,E1 24.9991,E2 -539.9392} C_DIS
LIN {X 0.488,Y -42.1896,Z 62,A -96.6446,B 24.8706,C -2.6249,E1 24.9991,E2 -539.9392} C_DIS
Enddeposition()
LIN {X 0.2272,Y -41.2107,Z 62,A -96.0832,B 24.8676,C -2.6551,E1 25.0009,E2 -540.5723} C_DIS
Startdeposition()
$VEL.CP = VEL_PRINT
LIN {X 2.7618,Y -41.1196,Z 62,A -91.358,B 24.8657,C -2.6738,E1 25.0142,E2 -545.3405} C_DIS
LIN {X 5.3426,Y -40.8645,Z 62,A -88.2428,B 24.8663,C -2.6686,E1 25.0228,E2 -548.4412} C_DIS
LIN {X 7.0817,Y -40.5991,Z 62,A -85.8542,B 24.8662,C -2.6696,E1 25.0294,E2 -550.8297} C_DIS
LIN {X 8.7932,Y -40.2632,Z 62,A -83.5315,B 24.8662,C -2.6701,E1 25.0357,E2 -553.1507} C_DIS
LIN {X 10.2853,Y -39.9082,Z 62,A -81.3441,B 24.8658,C -2.673,E1 25.0417,E2 -555.3419} C_DIS
LIN {X 11.818,Y -39.4816,Z 62,A -78.9562,B 24.8653,C -2.6781,E1 25.0481,E2 -557.7378} C_DIS
LIN {X 13.8147,Y -38.8283,Z 62,A -76.1587,B 24.8651,C -2.6798,E1 25.0555,E2 -560.5338} C_DIS
LIN {X 15.4329,Y -38.2136,Z 62,A -73.5193,B 24.8644,C -2.6867,E1 25.0624,E2 -563.1837} C_DIS
LIN {X 17.3521,Y -37.3812,Z 62,A -70.8911,B 24.8644,C -2.6867,E1 25.069,E2 -565.8053} C_DIS
LIN {X 19.1133,Y -36.5122,Z 62,A -67.9201,B 24.8636,C -2.6949,E1 25.0765,E2 -568.7877} C_DIS
LIN {X 20.7566,Y -35.6043,Z 62,A -65.6465,B 24.8636,C -2.6941,E1 25.082,E2 -571.0525} C_DIS
LIN {X 22.6951,Y -34.4003,Z 62,A -61.8101,B 24.862,C -2.7108,E1 25.091,E2 -574.9161} C_DIS
LIN {X 24.6559,Y -33.0235,Z 62,A -59.0055,B 24.8622,C -2.709,E1 25.0973,E2 -577.7065} C_DIS
LIN {X 25.9213,Y -32.0389,Z 62,A -56.4979,B 24.8612,C -2.7183,E1 25.1028,E2 -580.2267} C_DIS
LIN {X 28.4184,Y -29.8481,Z 62,A -51.3393,B 24.8592,C -2.7378,E1 25.1135,E2 -585.4108} C_DIS
LIN {X 31.4605,Y -26.6215,Z 62,A -46.3507,B 24.8597,C -2.7333,E1 25.1228,E2 -590.3666} C_DIS
LIN {X 33.0865,Y -24.5715,Z 62,A -41.7736,B 24.8571,C -2.7587,E1 25.1307,E2 -594.9821} C_DIS
LIN {X 34.7519,Y -22.1534,Z 62,A -38.0709,B 24.8566,C -2.7634,E1 25.1363,E2 -598.6775} C_DIS
LIN {X 36.176,Y -19.742,Z 62,A -34.7228,B 24.8564,C -2.7651,E1 25.141,E2 -602.0124} C_DIS
LIN {X 36.8197,Y -18.5152,Z 62,A -32.5392,B 24.8553,C -2.7751,E1 25.1437,E2 -604.2079} C_DIS
LIN {X 37.6964,Y -16.6573,Z 62,A -29.7985,B 24.8547,C -2.7815,E1 25.1469,E2 -606.9489} C_DIS
LIN {X 38.4937,Y -14.7208,Z 62,A -26.6462,B 24.8533,C -2.7944,E1 25.1502,E2 -610.1143} C_DIS
LIN {X 39.2254,Y -12.6418,Z 62,A -23.6809,B 24.8525,C -2.802,E1 25.1528,E2 -613.0809} C_DIS
LIN {X 39.8556,Y -10.4897,Z 62,A -20.5253,B 24.8514,C -2.8123,E1 25.1552,E2 -616.2426} C_DIS
LIN {X 40.4459,Y -7.9113,Z 62,A -17.185,B 24.8508,C -2.8179,E1 25.1571,E2 -619.5767} C_DIS
LIN {X 40.7535,Y -6.1341,Z 62,A -14.3111,B 24.8493,C -2.8321,E1 25.1584,E2 -622.4674} C_DIS
LIN {X 41.0734,Y -3.3818,Z 62,A -10.9659,B 24.849,C -2.8354,E1 25.1593,E2 -625.8006} C_DIS
LIN {X 41.1987,Y -1.0744,Z 62,A -6.9117,B 24.8463,C -2.8601,E1 25.1598,E2 -629.8892} C_DIS
LIN {X 41.1629,Y 2.0304,Z 62,A -3.3585,B 24.8463,C -2.8603,E1 25.1595,E2 -633.4217} C_DIS
LIN {X 40.9532,Y 4.608,Z 62,A 0.5396,B 24.8445,C -2.8767,E1 25.1585,E2 -637.3355} C_DIS
LIN {X 40.5307,Y 7.4605,Z 62,A 4.942,B 24.8424,C -2.8958,E1 25.1564,E2 -641.7572} C_DIS
LIN {X 39.8499,Y 10.5114,Z 62,A 8.5277,B 24.8424,C -2.8957,E1 25.1541,E2 -645.3219} C_DIS
LIN {X 39.3322,Y 12.3055,Z 62,A 11.0745,B 24.8417,C -2.9025,E1 25.152,E2 -647.8703} C_DIS
LIN {X 38.7657,Y 13.9889,Z 62,A 13.6569,B 24.8407,C -2.9116,E1 25.1496,E2 -650.4597} C_DIS
LIN {X 38.0771,Y 15.7677,Z 62,A 16.458,B 24.8396,C -2.9216,E1 25.1467,E2 -653.269} C_DIS
LIN {X 37.011,Y 18.1294,Z 62,A 19.6268,B 24.8393,C -2.9242,E1 25.143,E2 -656.4268} C_DIS
LIN {X 36.2398,Y 19.6247,Z 62,A 22.0998,B 24.8384,C -2.9327,E1 25.1397,E2 -658.907} C_DIS
LIN {X 35.4002,Y 21.102,Z 62,A 24.4138,B 24.8378,C -2.938,E1 25.1365,E2 -661.2217} C_DIS
LIN {X 33.95,Y 23.3641,Z 62,A 28.4281,B 24.8362,C -2.952,E1 25.1303,E2 -665.2491} C_DIS
LIN {X 32.4105,Y 25.4561,Z 62,A 32.0321,B 24.8353,C -2.9605,E1 25.1242,E2 -668.856} C_DIS
LIN {X 30.8011,Y 27.3817,Z 62,A 35.2811,B 24.8349,C -2.9644,E1 25.1183,E2 -672.0995} C_DIS
LIN {X 29.3924,Y 28.8885,Z 62,A 38.3402,B 24.8338,C -2.9735,E1 25.1123,E2 -675.1672} C_DIS
LIN {X 27.2934,Y 30.88,Z 62,A 42.2552,B 24.8331,C -2.9797,E1 25.1043,E2 -679.0809} C_DIS
LIN {X 25.6626,Y 32.2475,Z 62,A 45.3517,B 24.8323,C -2.9873,E1 25.0976,E2 -682.1837} C_DIS
LIN {X 23.1985,Y 34.063,Z 62,A 49.4967,B 24.8317,C -2.9926,E1 25.0882,E2 -686.3268} C_DIS
LIN {X 20.3748,Y 35.8228,Z 62,A 54.3166,B 24.8306,C -3.0023,E1 25.0766,E2 -691.1548} C_DIS
LIN {X 18.1699,Y 36.9908,Z 62,A 57.577,B 24.8305,C -3.0034,E1 25.0685,E2 -694.4089} C_DIS
LIN {X 16.0519,Y 37.9577,Z 62,A 61.2959,B 24.8292,C -3.0142,E1 25.0589,E2 -698.1444} C_DIS
LIN {X 13.4125,Y 38.9691,Z 62,A 64.4657,B 24.8301,C -3.0063,E1 25.0507,E2 -701.2889} C_DIS
LIN {X 11.0458,Y 39.7045,Z 62,A 68.6089,B 24.8287,C -3.0189,E1 25.0395,E2 -705.4551} C_DIS
LIN {X 8.7087,Y 40.2817,Z 62,A 72.1015,B 24.8283,C -3.0227,E1 25.03,E2 -708.952} C_DIS
LIN {X 4.4818,Y 40.9683,Z 62,A 77.9646,B 24.8283,C -3.0227,E1 25.0138,E2 -714.8103} C_DIS
LIN {X 0.7428,Y 41.2055,Z 62,A 82.6075,B 24.8292,C -3.0145,E1 25.0009,E2 -719.4322} C_DIS
LIN {X -2.2996,Y 41.148,Z 62,A 87.181,B 24.8288,C -3.0179,E1 24.9881,E2 -724.0146} C_DIS
LIN {X -4.9861,Y 40.9099,Z 62,A 90.6044,B 24.8295,C -3.0116,E1 24.9786,E2 -727.4248} C_DIS
LIN {X -7.1234,Y 40.5923,Z 62,A 93.4764,B 24.83,C -3.0077,E1 24.9707,E2 -730.2904} C_DIS
LIN {X -9.8891,Y 40.0084,Z 62,A 98.302,B 24.829,C -3.016,E1 24.9575,E2 -735.142} C_DIS
LIN {X -12.4374,Y 39.2912,Z 62,A 101.4985,B 24.8302,C -3.0056,E1 24.9491,E2 -738.3193} C_DIS
LIN {X -15.2349,Y 38.2927,Z 62,A 105.5156,B 24.831,C -2.9989,E1 24.9386,E2 -742.3287} C_DIS
LIN {X -16.9648,Y 37.5586,Z 62,A 108.0517,B 24.8315,C -2.9942,E1 24.9321,E2 -744.8596} C_DIS
LIN {X -18.8572,Y 36.6452,Z 62,A 111.0384,B 24.8319,C -2.9904,E1 24.9247,E2 -747.8452} C_DIS
LIN {X -21.2812,Y 35.2928,Z 62,A 114.2948,B 24.8335,C -2.9764,E1 24.9168,E2 -751.0777} C_DIS
LIN {X -23.7549,Y 33.6774,Z 62,A 119.752,B 24.8326,C -2.9848,E1 24.9041,E2 -756.5733} C_DIS
LIN {X -26.1118,Y 31.8852,Z 62,A 122.7764,B 24.835,C -2.9631,E1 24.8976,E2 -759.5572} C_DIS
LIN {X -27.5249,Y 30.673,Z 62,A 125.758,B 24.8351,C -2.962,E1 24.8913,E2 -762.5478} C_DIS
LIN {X -28.859,Y 29.4215,Z 62,A 128.3426,B 24.8357,C -2.9566,E1 24.8861,E2 -765.1303} C_DIS
LIN {X -30.1797,Y 28.0637,Z 62,A 130.917,B 24.8365,C -2.9496,E1 24.8812,E2 -767.6992} C_DIS
LIN {X -31.7981,Y 26.2175,Z 62,A 133.9853,B 24.8379,C -2.9371,E1 24.8757,E2 -770.7516} C_DIS
LIN {X -32.6501,Y 25.1479,Z 62,A 136.0777,B 24.8382,C -2.9343,E1 24.8721,E2 -772.8473} C_DIS
LIN {X -33.7017,Y 23.7212,Z 62,A 138.8364,B 24.8386,C -2.9311,E1 24.8676,E2 -775.6116} C_DIS
LIN {X -35.2036,Y 21.4279,Z 62,A 142.1285,B 24.8403,C -2.9149,E1 24.8627,E2 -778.8815} C_DIS
LIN {X -36.0683,Y 19.9384,Z 62,A 144.738,B 24.8408,C -2.9105,E1 24.8591,E2 -781.4942} C_DIS
LIN {X -36.7925,Y 18.5688,Z 62,A 147.0456,B 24.8413,C -2.906,E1 24.8561,E2 -783.8034} C_DIS
LIN {X -37.8489,Y 16.3077,Z 62,A 150.6642,B 24.8423,C -2.8975,E1 24.852,E2 -787.4215} C_DIS
LIN {X -39.0275,Y 13.2402,Z 62,A 155.5273,B 24.8434,C -2.8869,E1 24.8473,E2 -792.2868} C_DIS
LIN {X -39.6819,Y 11.1269,Z 62,A 158.8185,B 24.8442,C -2.8799,E1 24.8448,E2 -795.5802} C_DIS
LIN {X -40.4849,Y 7.709,Z 62,A 163.3175,B 24.8463,C -2.8605,E1 24.8422,E2 -800.0594} C_DIS
LIN {X -40.8977,Y 5.0769,Z 62,A 166.6598,B 24.8479,C -2.8451,E1 24.8408,E2 -803.3846} C_DIS
LIN {X -41.0583,Y 3.5651,Z 62,A 169.1388,B 24.8482,C -2.8424,E1 24.8402,E2 -805.872} C_DIS
LIN {X -41.1953,Y 1.1837,Z 62,A 172.5407,B 24.8492,C -2.8329,E1 24.8398,E2 -809.2717} C_DIS
LIN {X -41.2069,Y -0.6662,Z 62,A 175.2492,B 24.8499,C -2.8264,E1 24.8398,E2 -811.9809} C_DIS
LIN {X -41.1112,Y -2.8863,Z 62,A 177.8723,B 24.8515,C -2.8117,E1 24.8403,E2 -814.5846} C_DIS
LIN {X -40.98,Y -4.3699,Z 62,A 179.8616,B 24.8523,C -2.8044,E1 24.8408,E2 -816.5684} C_DIS
LIN {X -40.698,Y -6.4931,Z 62,A -176.4953,B 24.8525,C -2.8025,E1 24.8423,E2 -820.2287} C_DIS
LIN {X -40.2345,Y -8.925,Z 62,A -173.4088,B 24.854,C -2.7882,E1 24.844,E2 -823.2992} C_DIS
LIN {X -39.764,Y -10.8296,Z 62,A -170.5353,B 24.8547,C -2.7817,E1 24.8461,E2 -826.174} C_DIS
LIN {X -39.0908,Y -13.0522,Z 62,A -166.9933,B 24.8553,C -2.7758,E1 24.8491,E2 -829.7221} C_DIS
LIN {X -38.0871,Y -15.744,Z 62,A -163.0495,B 24.8565,C -2.7639,E1 24.8531,E2 -833.6595} C_DIS
LIN {X -36.8712,Y -18.4113,Z 62,A -159.4186,B 24.8582,C -2.7477,E1 24.8575,E2 -837.2715} C_DIS
LIN {X -35.9346,Y -20.1782,Z 62,A -156.3593,B 24.8586,C -2.7435,E1 24.8616,E2 -840.3369} C_DIS
LIN {X -34.5984,Y -22.3925,Z 62,A -153.3387,B 24.8603,C -2.7278,E1 24.866,E2 -843.3352} C_DIS
LIN {X -33.153,Y -24.4807,Z 62,A -149.4087,B 24.8607,C -2.7238,E1 24.8723,E2 -847.275} C_DIS
LIN {X -31.7421,Y -26.2848,Z 62,A -145.5769,B 24.8607,C -2.7241,E1 24.879,E2 -851.1255} C_DIS
LIN {X -29.9369,Y -28.324,Z 62,A -141.8776,B 24.8616,C -2.7149,E1 24.886,E2 -854.8191} C_DIS
LIN {X -27.8247,Y -30.4012,Z 62,A -138.0762,B 24.8628,C -2.7028,E1 24.8937,E2 -858.6073} C_DIS
LIN {X -25.9402,Y -32.0242,Z 62,A -134.6005,B 24.8634,C -2.6967,E1 24.9012,E2 -862.0817} C_DIS
LIN {X -23.2688,Y -34.0148,Z 62,A -129.6172,B 24.8638,C -2.6935,E1 24.9125,E2 -867.0746} C_DIS
LIN {X -21.2199,Y -35.3294,Z 62,A -126.4431,B 24.8645,C -2.6859,E1 24.92,E2 -870.2405} C_DIS
LIN {X -19.0027,Y -36.5705,Z 62,A -122.406,B 24.8643,C -2.6879,E1 24.93,E2 -874.2938} C_DIS
LIN {X -16.353,Y -37.8291,Z 62,A -119.1255,B 24.8658,C -2.673,E1 24.9383,E2 -877.5467} C_DIS
Enddeposition()
END
